LIN {X 0,Y 262.413,Z 305.616,A -85,B 0,C 180,E1 -18658.413,E2 -18658.413} C_VEL
LIN {X 0,Y 260.939,Z 356.529,A -85,B 0,C 180,E1 -18660.058,E2 -18660.058} C_VEL
LIN {X 0,Y 260.58,Z 366.415,A -85,B 0,C 180,E1 -18660.585,E2 -18660.585} C_VEL
LIN {X 0,Y 259.89,Z 377.928,A -85,B 0,C 180,E1 -18661.482,E2 -18661.482} C_VEL
LIN {X 0,Y 259.092,Z 388.369,A -85,B 0,C 180,E1 -18662.636,E2 -18662.636} C_VEL
LIN {X 0,Y 258.368,Z 397.253,A -85,B 0,C 180,E1 -18663.891,E2 -18663.891} C_VEL
LIN {X 0,Y 257.495,Z 404.951,A -85,B 0,C 180,E1 -18665.226,E2 -18665.226} C_VEL
LIN {X 0,Y 256.533,Z 413.514,A -85,B 0,C 180,E1 -18667.063,E2 -18667.063} C_VEL
LIN {X 0,Y 255.727,Z 421.136,A -85,B 0,C 180,E1 -18669.203,E2 -18669.203} C_VEL
LIN {X 0,Y 255.116,Z 426.116,A -85,B 0,C 180,E1 -18670.941,E2 -18670.941} C_VEL
LIN {X 0,Y 254.737,Z 430.48,A -85,B 0,C 180,E1 -18672.842,E2 -18672.842} C_VEL
LIN {X 0,Y 254.278,Z 434.421,A -85,B 0,C 180,E1 -18675.095,E2 -18675.095} C_VEL
LIN {X 0,Y 254.025,Z 437.165,A -85,B 0,C 180,E1 -18677.329,E2 -18677.329} C_VEL
LIN {X 0,Y 254.008,Z 438.048,A -85,B 0,C 180,E1 -18678.393,E2 -18678.393} C_VEL
LIN {X 0,Y 254.169,Z 439.211,A -85,B 0,C 180,E1 -18680.733,E2 -18680.733} C_VEL
LIN {X 0,Y 254.592,Z 439.262,A -85,B 0,C 180,E1 -18683.18,E2 -18683.18} C_VEL
LIN {X 0,Y 255.349,Z 438.101,A -85,B 0,C 180,E1 -18685.656,E2 -18685.656} C_VEL
LIN {X 0,Y 256.573,Z 434.825,A -85,B 0,C 180,E1 -18688.64,E2 -18688.64} C_VEL
LIN {X 0,Y 257.683,Z 431.567,A -85,B 0,C 180,E1 -18690.6,E2 -18690.6} C_VEL
LIN {X 0,Y 258.955,Z 427.356,A -85,B 0,C 180,E1 -18692.526,E2 -18692.526} C_VEL
LIN {X 0,Y 260.481,Z 422.037,A -85,B 0,C 180,E1 -18694.427,E2 -18694.427} C_VEL
LIN {X 0,Y 262.359,Z 415.32,A -85,B 0,C 180,E1 -18696.31,E2 -18696.31} C_VEL
LIN {X 0,Y 264.289,Z 406.845,A -85,B 0,C 180,E1 -18698.145,E2 -18698.145} C_VEL
LIN {X 0,Y 265.906,Z 399.02,A -85,B 0,C 180,E1 -18699.502,E2 -18699.502} C_VEL
LIN {X 0,Y 267.227,Z 391.67,A -85,B 0,C 180,E1 -18700.543,E2 -18700.543} C_VEL
LIN {X 0,Y 268.577,Z 382.564,A -85,B 0,C 180,E1 -18701.58,E2 -18701.58} C_VEL
LIN {X 0,Y 269.878,Z 372.132,A -85,B 0,C 180,E1 -18702.478,E2 -18702.478} C_VEL
LIN {X 0,Y 270.737,Z 360.477,A -85,B 0,C 180,E1 -18703.167,E2 -18703.167} C_VEL
LIN {X 0,Y 271.796,Z 338.049,A -85,B 0,C 180,E1 -18703.941,E2 -18703.941} C_VEL
LIN {X 0,Y 272.811,Z 314.84,A -85,B 0,C 180,E1 -18704.695,E2 -18704.695} C_VEL
LIN {X 0,Y 268.494,Z 305.093,A -85,B 0,C 180,E1 -18705.731,E2 -18705.731} C_VEL
LIN {X 0,Y 262.601,Z 294.531,A -85,B 0,C 180,E1 -18707.147,E2 -18707.147} C_VEL
LIN {X 0,Y 258.247,Z 287.429,A -85,B 0,C 180,E1 -18708.241,E2 -18708.241} C_VEL
LIN {X 0,Y 256.704,Z 285.058,A -85,B 0,C 180,E1 -18708.638,E2 -18708.638} C_VEL
LIN {X 0,Y 256.281,Z 283.378,A -85,B 0,C 180,E1 -18708.844,E2 -18708.844} C_VEL
LIN {X 0,Y 256.508,Z 283.344,A -85,B 0,C 180,E1 -18712.128,E2 -18712.128} C_VEL
LIN {X 0,Y 256.494,Z 283.345,A -85,B 0,C 180,E1 -18716.86,E2 -18716.86} C_VEL
LIN {X 0,Y 256.759,Z 283.312,A -85,B 0,C 180,E1 -18720.001,E2 -18720.001} C_VEL
LIN {X 0,Y 256.494,Z 283.347,A -85,B 0,C 180,E1 -18723.143,E2 -18723.143} C_VEL
LIN {X 0,Y 256.534,Z 283.334,A -85,B 0,C 180,E1 -18727.874,E2 -18727.874} C_VEL
LIN {X 0,Y 256.503,Z 283.337,A -85,B 0,C 180,E1 -18728.248,E2 -18728.248} C_VEL
LIN {X 0,Y 255.757,Z 283.436,A -85,B 0,C 180,E1 -18729.556,E2 -18729.556} C_VEL
LIN {X 0,Y 252.8,Z 283.81,A -85,B 0,C 180,E1 -18731.686,E2 -18731.686} C_VEL
LIN {X 0,Y 250.323,Z 284.12,A -85,B 0,C 180,E1 -18733.42,E2 -18733.42} C_VEL
LIN {X 0,Y 249.264,Z 284.248,A -85,B 0,C 180,E1 -18734.766,E2 -18734.766} C_VEL
LIN {X 0,Y 249.178,Z 284.253,A -85,B 0,C 180,E1 -18735.223,E2 -18735.223} C_VEL
LIN {X 0,Y 249.131,Z 284.26,A -85,B 0,C 180,E1 -18738.079,E2 -18738.079} C_VEL
LIN {X 0,Y 249.084,Z 284.258,A -85,B 0,C 180,E1 -18741.52,E2 -18741.52} C_VEL
LIN {X 0,Y 249.128,Z 284.252,A -85,B 0,C 180,E1 -18745.484,E2 -18745.484} C_VEL
LIN {X 0,Y 249.083,Z 284.259,A -85,B 0,C 180,E1 -18748.996,E2 -18748.996} C_VEL
LIN {X 0,Y 249.034,Z 284.271,A -85,B 0,C 180,E1 -18752.427,E2 -18752.427} C_VEL
LIN {X 0,Y 249.072,Z 284.267,A -85,B 0,C 180,E1 -18756.339,E2 -18756.339} C_VEL
LIN {X 0,Y 249.036,Z 284.27,A -85,B 0,C 180,E1 -18760.473,E2 -18760.473} C_VEL
LIN {X 0,Y 249.033,Z 284.276,A -85,B 0,C 180,E1 -18762.8,E2 -18762.8} C_VEL
LIN {X 0,Y 249.018,Z 284.277,A -85,B 0,C 180,E1 -18767.365,E2 -18767.365} C_VEL
LIN {X 0,Y 249.056,Z 284.41,A -85,B 0,C 180,E1 -18771.174,E2 -18771.174} C_VEL
LIN {X 0,Y 250.877,Z 290.539,A -85,B 0,C 180,E1 -18774.332,E2 -18774.332} C_VEL
LIN {X 0,Y 252.867,Z 298.716,A -85,B 0,C 180,E1 -18778.126,E2 -18778.126} C_VEL
LIN {X 0,Y 253.754,Z 302.564,A -85,B 0,C 180,E1 -18779.725,E2 -18779.725} C_VEL
LIN {X 0,Y 255.811,Z 306.867,A -85,B 0,C 180,E1 -18780.308,E2 -18780.308} C_VEL
LIN {X 0,Y 259.48,Z 315.185,A -85,B 0,C 180,E1 -18781.332,E2 -18781.332} C_VEL
LIN {X 0,Y 262.764,Z 332.237,A -85,B 0,C 180,E1 -18782.601,E2 -18782.601} C_VEL
LIN {X 0,Y 264.983,Z 349.14,A -85,B 0,C 180,E1 -18783.635,E2 -18783.635} C_VEL
LIN {X 0,Y 265.432,Z 356.335,A -85,B 0,C 180,E1 -18783.987,E2 -18783.987} C_VEL
LIN {X 0,Y 263.95,Z 383.888,A -85,B 0,C 180,E1 -18784.924,E2 -18784.924} C_VEL
LIN {X 0,Y 262.737,Z 395.64,A -85,B 0,C 180,E1 -18785.573,E2 -18785.573} C_VEL
LIN {X 0,Y 261.153,Z 405.827,A -85,B 0,C 180,E1 -18786.404,E2 -18786.404} C_VEL
LIN {X 0,Y 259.584,Z 414.308,A -85,B 0,C 180,E1 -18787.307,E2 -18787.307} C_VEL
LIN {X 0,Y 257.892,Z 422.523,A -85,B 0,C 180,E1 -18788.415,E2 -18788.415} C_VEL
LIN {X 0,Y 256.092,Z 430.382,A -85,B 0,C 180,E1 -18789.729,E2 -18789.729} C_VEL
LIN {X 0,Y 254.423,Z 436.939,A -85,B 0,C 180,E1 -18791.061,E2 -18791.061} C_VEL
LIN {X 0,Y 252.738,Z 443.225,A -85,B 0,C 180,E1 -18792.607,E2 -18792.607} C_VEL
LIN {X 0,Y 251.217,Z 448.504,A -85,B 0,C 180,E1 -18794.172,E2 -18794.172} C_VEL
LIN {X 0,Y 249.775,Z 453.917,A -85,B 0,C 180,E1 -18796.163,E2 -18796.163} C_VEL
LIN {X 0,Y 248.415,Z 459.006,A -85,B 0,C 180,E1 -18798.578,E2 -18798.578} C_VEL
LIN {X 0,Y 247.812,Z 461.526,A -85,B 0,C 180,E1 -18800.203,E2 -18800.203} C_VEL
LIN {X 0,Y 247.369,Z 463.503,A -85,B 0,C 180,E1 -18801.834,E2 -18801.834} C_VEL
LIN {X 0,Y 246.986,Z 465.878,A -85,B 0,C 180,E1 -18804.834,E2 -18804.834} C_VEL
LIN {X 0,Y 247.05,Z 466.43,A -85,B 0,C 180,E1 -18806.739,E2 -18806.739} C_VEL
LIN {X 0,Y 247.107,Z 466.306,A -85,B 0,C 180,E1 -18808.371,E2 -18808.371} C_VEL
LIN {X 0,Y 247.233,Z 465.701,A -85,B 0,C 180,E1 -18810,E2 -18810} C_VEL
LIN {X 0,Y 247.156,Z 464.577,A -85,B 0,C 180,E1 -18811.63,E2 -18811.63} C_VEL
LIN {X 0,Y 247.203,Z 462.925,A -85,B 0,C 180,E1 -18813.26,E2 -18813.26} C_VEL
LIN {X 0,Y 247.195,Z 459.237,A -85,B 0,C 180,E1 -18815.676,E2 -18815.676} C_VEL
LIN {X 0,Y 247.425,Z 453.965,A -85,B 0,C 180,E1 -18818.165,E2 -18818.165} C_VEL
LIN {X 0,Y 247.837,Z 448.329,A -85,B 0,C 180,E1 -18820.209,E2 -18820.209} C_VEL
LIN {X 0,Y 248.555,Z 441.204,A -85,B 0,C 180,E1 -18822.244,E2 -18822.244} C_VEL
LIN {X 0,Y 249.399,Z 433.015,A -85,B 0,C 180,E1 -18824.067,E2 -18824.067} C_VEL
LIN {X 0,Y 250.162,Z 426.449,A -85,B 0,C 180,E1 -18825.271,E2 -18825.271} C_VEL
LIN {X 0,Y 250.921,Z 420.034,A -85,B 0,C 180,E1 -18826.266,E2 -18826.266} C_VEL
LIN {X 0,Y 251.602,Z 412.242,A -85,B 0,C 180,E1 -18827.265,E2 -18827.265} C_VEL
LIN {X 0,Y 252.641,Z 402.367,A -85,B 0,C 180,E1 -18828.237,E2 -18828.237} C_VEL
LIN {X 0,Y 253.32,Z 393.113,A -85,B 0,C 180,E1 -18828.92,E2 -18828.92} C_VEL
LIN {X 0,Y 253.729,Z 383.59,A -85,B 0,C 180,E1 -18829.414,E2 -18829.414} C_VEL
LIN {X 0,Y 254.605,Z 351.161,A -85,B 0,C 180,E1 -18830.505,E2 -18830.505} C_VEL
LIN {X 0,Y 250.337,Z 306.801,A -85,B 0,C 180,E1 -18832.309,E2 -18832.309} C_VEL
LIN {X 0,Y 251.565,Z 297.448,A -85,B 0,C 180,E1 -18835.66,E2 -18835.66} C_VEL
LIN {X 0,Y 249.84,Z 287.931,A -85,B 0,C 180,E1 -18839.303,E2 -18839.303} C_VEL
LIN {X 0,Y 249.12,Z 284.266,A -85,B 0,C 180,E1 -18840.752,E2 -18840.752} C_VEL
LIN {X 0,Y 249.052,Z 284.273,A -85,B 0,C 180,E1 -18845.079,E2 -18845.079} C_VEL
LIN {X 0,Y 249.04,Z 284.274,A -85,B 0,C 180,E1 -18848.378,E2 -18848.378} C_VEL
LIN {X 0,Y 249.014,Z 284.275,A -85,B 0,C 180,E1 -18852.792,E2 -18852.792} C_VEL
LIN {X 0,Y 249.011,Z 284.28,A -85,B 0,C 180,E1 -18857.36,E2 -18857.36} C_VEL
LIN {X 0,Y 249.026,Z 284.277,A -85,B 0,C 180,E1 -18861.618,E2 -18861.618} C_VEL
LIN {X 0,Y 249.044,Z 284.277,A -85,B 0,C 180,E1 -18865.638,E2 -18865.638} C_VEL
LIN {X 0,Y 249.052,Z 284.274,A -85,B 0,C 180,E1 -18869.472,E2 -18869.472} C_VEL
LIN {X 0,Y 249.074,Z 284.271,A -85,B 0,C 180,E1 -18873.161,E2 -18873.161} C_VEL
LIN {X 0,Y 249.079,Z 284.268,A -85,B 0,C 180,E1 -18876.731,E2 -18876.731} C_VEL
LIN {X 0,Y 249.11,Z 284.265,A -85,B 0,C 180,E1 -18880.21,E2 -18880.21} C_VEL
LIN {X 0,Y 249.241,Z 284.253,A -85,B 0,C 180,E1 -18883.621,E2 -18883.621} C_VEL
LIN {X 0,Y 249.242,Z 284.247,A -85,B 0,C 180,E1 -18888.615,E2 -18888.615} C_VEL
LIN {X 0,Y 249.453,Z 284.224,A -85,B 0,C 180,E1 -18891.901,E2 -18891.901} C_VEL
LIN {X 0,Y 249.294,Z 284.241,A -85,B 0,C 180,E1 -18895.147,E2 -18895.147} C_VEL
LIN {X 0,Y 249.673,Z 284.195,A -85,B 0,C 180,E1 -18898.386,E2 -18898.386} C_VEL
LIN {X 0,Y 249.673,Z 284.199,A -85,B 0,C 180,E1 -18901.612,E2 -18901.612} C_VEL
LIN {X 0,Y 249.446,Z 284.221,A -85,B 0,C 180,E1 -18906.773,E2 -18906.773} C_VEL
LIN {X 0,Y 249.385,Z 284.234,A -85,B 0,C 180,E1 -18909.733,E2 -18909.733} C_VEL
LIN {X 0,Y 249.197,Z 284.253,A -85,B 0,C 180,E1 -18914.702,E2 -18914.702} C_VEL
LIN {X 0,Y 249.135,Z 284.263,A -85,B 0,C 180,E1 -18918.076,E2 -18918.076} C_VEL
LIN {X 0,Y 249.099,Z 284.267,A -85,B 0,C 180,E1 -18921.515,E2 -18921.515} C_VEL
LIN {X 0,Y 249.125,Z 284.266,A -85,B 0,C 180,E1 -18925.481,E2 -18925.481} C_VEL
LIN {X 0,Y 249.075,Z 284.268,A -85,B 0,C 180,E1 -18928.991,E2 -18928.991} C_VEL
LIN {X 0,Y 249.03,Z 284.275,A -85,B 0,C 180,E1 -18932.424,E2 -18932.424} C_VEL
LIN {X 0,Y 249.07,Z 284.269,A -85,B 0,C 180,E1 -18936.337,E2 -18936.337} C_VEL
LIN {X 0,Y 249.032,Z 284.275,A -85,B 0,C 180,E1 -18940.471,E2 -18940.471} C_VEL
LIN {X 0,Y 249.042,Z 284.273,A -85,B 0,C 180,E1 -18942.801,E2 -18942.801} C_VEL
LIN {X 0,Y 249.056,Z 284.271,A -85,B 0,C 180,E1 -18947.372,E2 -18947.372} C_VEL
LIN {X 0,Y 249.046,Z 284.277,A -85,B 0,C 180,E1 -18951.623,E2 -18951.623} C_VEL
LIN {X 0,Y 249.055,Z 284.273,A -85,B 0,C 180,E1 -18955.642,E2 -18955.642} C_VEL
LIN {X 0,Y 249.045,Z 284.275,A -85,B 0,C 180,E1 -18959.472,E2 -18959.472} C_VEL
LIN {X 0,Y 249.067,Z 284.269,A -85,B 0,C 180,E1 -18963.162,E2 -18963.162} C_VEL
LIN {X 0,Y 249.072,Z 284.27,A -85,B 0,C 180,E1 -18966.732,E2 -18966.732} C_VEL
LIN {X 0,Y 249.103,Z 284.266,A -85,B 0,C 180,E1 -18970.211,E2 -18970.211} C_VEL
LIN {X 0,Y 249.235,Z 284.251,A -85,B 0,C 180,E1 -18973.621,E2 -18973.621} C_VEL
LIN {X 0,Y 249.246,Z 284.247,A -85,B 0,C 180,E1 -18978.616,E2 -18978.616} C_VEL
LIN {X 0,Y 249.474,Z 284.223,A -85,B 0,C 180,E1 -18981.902,E2 -18981.902} C_VEL
LIN {X 0,Y 249.426,Z 284.225,A -85,B 0,C 180,E1 -18986.769,E2 -18986.769} C_VEL
LIN {X 0,Y 249.72,Z 284.191,A -85,B 0,C 180,E1 -18990,E2 -18990} C_VEL
LIN {X 0,Y 249.426,Z 284.226,A -85,B 0,C 180,E1 -18993.23,E2 -18993.23} C_VEL
LIN {X 0,Y 249.472,Z 284.221,A -85,B 0,C 180,E1 -18998.097,E2 -18998.097} C_VEL
LIN {X 0,Y 249.245,Z 284.249,A -85,B 0,C 180,E1 -19001.383,E2 -19001.383} C_VEL
LIN {X 0,Y 249.234,Z 284.251,A -85,B 0,C 180,E1 -19006.378,E2 -19006.378} C_VEL
LIN {X 0,Y 249.076,Z 284.272,A -85,B 0,C 180,E1 -19011.518,E2 -19011.518} C_VEL
LIN {X 0,Y 249.112,Z 284.267,A -85,B 0,C 180,E1 -19015.477,E2 -19015.477} C_VEL
LIN {X 0,Y 249.137,Z 284.413,A -85,B 0,C 180,E1 -19016.89,E2 -19016.89} C_VEL
LIN {X 0,Y 255.379,Z 303.773,A -85,B 0,C 180,E1 -19017.949,E2 -19017.949} C_VEL
LIN {X 0,Y 255.335,Z 313.119,A -85,B 0,C 180,E1 -19018.266,E2 -19018.266} C_VEL
LIN {X 0,Y 253.983,Z 356.955,A -85,B 0,C 180,E1 -19019.729,E2 -19019.729} C_VEL
LIN {X 0,Y 253.595,Z 367.606,A -85,B 0,C 180,E1 -19020.321,E2 -19020.321} C_VEL
LIN {X 0,Y 252.936,Z 378.268,A -85,B 0,C 180,E1 -19021.188,E2 -19021.188} C_VEL
LIN {X 0,Y 252.224,Z 387.215,A -85,B 0,C 180,E1 -19022.173,E2 -19022.173} C_VEL
LIN {X 0,Y 251.439,Z 396.631,A -85,B 0,C 180,E1 -19023.503,E2 -19023.503} C_VEL
LIN {X 0,Y 250.641,Z 403.843,A -85,B 0,C 180,E1 -19024.749,E2 -19024.749} C_VEL
LIN {X 0,Y 249.787,Z 410.867,A -85,B 0,C 180,E1 -19026.216,E2 -19026.216} C_VEL
LIN {X 0,Y 249.097,Z 417.185,A -85,B 0,C 180,E1 -19027.818,E2 -19027.818} C_VEL
LIN {X 0,Y 248.377,Z 423.251,A -85,B 0,C 180,E1 -19029.694,E2 -19029.694} C_VEL
LIN {X 0,Y 247.772,Z 429.196,A -85,B 0,C 180,E1 -19032.015,E2 -19032.015} C_VEL
LIN {X 0,Y 247.392,Z 432.744,A -85,B 0,C 180,E1 -19033.825,E2 -19033.825} C_VEL
LIN {X 0,Y 247.157,Z 435.002,A -85,B 0,C 180,E1 -19035.305,E2 -19035.305} C_VEL
LIN {X 0,Y 246.912,Z 437.829,A -85,B 0,C 180,E1 -19037.734,E2 -19037.734} C_VEL
LIN {X 0,Y 247.024,Z 439.415,A -85,B 0,C 180,E1 -19040.188,E2 -19040.188} C_VEL
LIN {X 0,Y 247.552,Z 439.696,A -85,B 0,C 180,E1 -19043.405,E2 -19043.405} C_VEL
LIN {X 0,Y 248.2,Z 438.833,A -85,B 0,C 180,E1 -19045.508,E2 -19045.508} C_VEL
LIN {X 0,Y 249.12,Z 436.904,A -85,B 0,C 180,E1 -19047.813,E2 -19047.813} C_VEL
LIN {X 0,Y 250.496,Z 433.299,A -85,B 0,C 180,E1 -19050.426,E2 -19050.426} C_VEL
LIN {X 0,Y 251.767,Z 429.419,A -85,B 0,C 180,E1 -19052.413,E2 -19052.413} C_VEL
LIN {X 0,Y 253.445,Z 423.975,A -85,B 0,C 180,E1 -19054.546,E2 -19054.546} C_VEL
LIN {X 0,Y 254.957,Z 418.94,A -85,B 0,C 180,E1 -19056.118,E2 -19056.118} C_VEL
LIN {X 0,Y 256.614,Z 412.846,A -85,B 0,C 180,E1 -19057.68,E2 -19057.68} C_VEL
LIN {X 0,Y 258.212,Z 406.364,A -85,B 0,C 180,E1 -19059.046,E2 -19059.046} C_VEL
LIN {X 0,Y 259.864,Z 398.652,A -85,B 0,C 180,E1 -19060.382,E2 -19060.382} C_VEL
LIN {X 0,Y 261.442,Z 390.014,A -85,B 0,C 180,E1 -19061.589,E2 -19061.589} C_VEL
LIN {X 0,Y 263.194,Z 378.281,A -85,B 0,C 180,E1 -19062.82,E2 -19062.82} C_VEL
LIN {X 0,Y 264.216,Z 367.992,A -85,B 0,C 180,E1 -19063.598,E2 -19063.598} C_VEL
LIN {X 0,Y 264.948,Z 358.296,A -85,B 0,C 180,E1 -19064.098,E2 -19064.098} C_VEL
LIN {X 0,Y 266.9,Z 316.919,A -85,B 0,C 180,E1 -19065.501,E2 -19065.501} C_VEL
LIN {X 0,Y 263.411,Z 308.95,A -85,B 0,C 180,E1 -19066.403,E2 -19066.403} C_VEL
LIN {X 0,Y 257.551,Z 298.407,A -85,B 0,C 180,E1 -19067.877,E2 -19067.877} C_VEL
LIN {X 0,Y 253.374,Z 291.754,A -85,B 0,C 180,E1 -19068.983,E2 -19068.983} C_VEL
LIN {X 0,Y 251.406,Z 288.478,A -85,B 0,C 180,E1 -19069.533,E2 -19069.533} C_VEL
LIN {X 0,Y 249.771,Z 285.962,A -85,B 0,C 180,E1 -19069.996,E2 -19069.996} C_VEL
LIN {X 0,Y 249.357,Z 284.236,A -85,B 0,C 180,E1 -19070.215,E2 -19070.215} C_VEL
LIN {X 0,Y 249.447,Z 284.228,A -85,B 0,C 180,E1 -19073.531,E2 -19073.531} C_VEL
LIN {X 0,Y 249.67,Z 284.193,A -85,B 0,C 180,E1 -19078.388,E2 -19078.388} C_VEL
LIN {X 0,Y 249.67,Z 284.191,A -85,B 0,C 180,E1 -19081.614,E2 -19081.614} C_VEL
LIN {X 0,Y 249.455,Z 284.226,A -85,B 0,C 180,E1 -19086.472,E2 -19086.472} C_VEL
LIN {X 0,Y 249.384,Z 284.232,A -85,B 0,C 180,E1 -19089.736,E2 -19089.736} C_VEL
LIN {X 0,Y 249.193,Z 284.257,A -85,B 0,C 180,E1 -19094.705,E2 -19094.705} C_VEL
LIN {X 0,Y 249.178,Z 284.253,A -85,B 0,C 180,E1 -19095.223,E2 -19095.223} C_VEL
LIN {X 0,Y 248.502,Z 284.332,A -85,B 0,C 180,E1 -19096.571,E2 -19096.571} C_VEL
LIN {X 0,Y 245.618,Z 284.702,A -85,B 0,C 180,E1 -19098.767,E2 -19098.767} C_VEL
LIN {X 0,Y 243.16,Z 285.008,A -85,B 0,C 180,E1 -19100.555,E2 -19100.555} C_VEL
LIN {X 0,Y 242.095,Z 285.134,A -85,B 0,C 180,E1 -19101.943,E2 -19101.943} C_VEL
LIN {X 0,Y 242.002,Z 285.144,A -85,B 0,C 180,E1 -19102.414,E2 -19102.414} C_VEL
LIN {X 0,Y 242.064,Z 285.133,A -85,B 0,C 180,E1 -19105.84,E2 -19105.84} C_VEL
LIN {X 0,Y 242.029,Z 285.137,A -85,B 0,C 180,E1 -19109.582,E2 -19109.582} C_VEL
LIN {X 0,Y 241.989,Z 285.143,A -85,B 0,C 180,E1 -19113.493,E2 -19113.493} C_VEL
LIN {X 0,Y 242.009,Z 285.143,A -85,B 0,C 180,E1 -19117.58,E2 -19117.58} C_VEL
LIN {X 0,Y 241.96,Z 285.158,A -85,B 0,C 180,E1 -19121.919,E2 -19121.919} C_VEL
LIN {X 0,Y 241.937,Z 285.156,A -85,B 0,C 180,E1 -19126.572,E2 -19126.572} C_VEL
LIN {X 0,Y 241.989,Z 285.359,A -85,B 0,C 180,E1 -19129.812,E2 -19129.812} C_VEL
LIN {X 0,Y 244.398,Z 293.32,A -85,B 0,C 180,E1 -19134.17,E2 -19134.17} C_VEL
LIN {X 0,Y 246.442,Z 301.873,A -85,B 0,C 180,E1 -19138.198,E2 -19138.198} C_VEL
LIN {X 0,Y 252.059,Z 313.372,A -85,B 0,C 180,E1 -19139.894,E2 -19139.894} C_VEL
LIN {X 0,Y 254.241,Z 318.686,A -85,B 0,C 180,E1 -19140.55,E2 -19140.55} C_VEL
LIN {X 0,Y 257.29,Z 334.984,A -85,B 0,C 180,E1 -19141.802,E2 -19141.802} C_VEL
LIN {X 0,Y 259.369,Z 352.201,A -85,B 0,C 180,E1 -19142.88,E2 -19142.88} C_VEL
LIN {X 0,Y 259.575,Z 357.239,A -85,B 0,C 180,E1 -19143.125,E2 -19143.125} C_VEL
LIN {X 0,Y 258.032,Z 383.822,A -85,B 0,C 180,E1 -19144.06,E2 -19144.06} C_VEL
LIN {X 0,Y 256.733,Z 395.495,A -85,B 0,C 180,E1 -19144.728,E2 -19144.728} C_VEL
LIN {X 0,Y 255.075,Z 405.756,A -85,B 0,C 180,E1 -19145.589,E2 -19145.589} C_VEL
LIN {X 0,Y 253.425,Z 414.174,A -85,B 0,C 180,E1 -19146.507,E2 -19146.507} C_VEL
LIN {X 0,Y 251.644,Z 422.342,A -85,B 0,C 180,E1 -19147.635,E2 -19147.635} C_VEL
LIN {X 0,Y 249.756,Z 430.165,A -85,B 0,C 180,E1 -19148.976,E2 -19148.976} C_VEL
LIN {X 0,Y 247.753,Z 437.555,A -85,B 0,C 180,E1 -19150.531,E2 -19150.531} C_VEL
LIN {X 0,Y 245.573,Z 445.112,A -85,B 0,C 180,E1 -19152.513,E2 -19152.513} C_VEL
LIN {X 0,Y 243.418,Z 452.074,A -85,B 0,C 180,E1 -19154.94,E2 -19154.94} C_VEL
LIN {X 0,Y 241.857,Z 457.428,A -85,B 0,C 180,E1 -19157.413,E2 -19157.413} C_VEL
LIN {X 0,Y 240.785,Z 461.439,A -85,B 0,C 180,E1 -19159.915,E2 -19159.915} C_VEL
LIN {X 0,Y 240.326,Z 463.323,A -85,B 0,C 180,E1 -19161.593,E2 -19161.593} C_VEL
LIN {X 0,Y 240.033,Z 464.71,A -85,B 0,C 180,E1 -19163.275,E2 -19163.275} C_VEL
LIN {X 0,Y 239.923,Z 465.624,A -85,B 0,C 180,E1 -19164.959,E2 -19164.959} C_VEL
LIN {X 0,Y 239.962,Z 466.046,A -85,B 0,C 180,E1 -19166.642,E2 -19166.642} C_VEL
LIN {X 0,Y 240.032,Z 465.859,A -85,B 0,C 180,E1 -19168.323,E2 -19168.323} C_VEL
LIN {X 0,Y 240.152,Z 465.168,A -85,B 0,C 180,E1 -19170,E2 -19170} C_VEL
LIN {X 0,Y 240.084,Z 463.96,A -85,B 0,C 180,E1 -19171.678,E2 -19171.678} C_VEL
LIN {X 0,Y 240.141,Z 462.229,A -85,B 0,C 180,E1 -19173.356,E2 -19173.356} C_VEL
LIN {X 0,Y 240.109,Z 458.853,A -85,B 0,C 180,E1 -19175.618,E2 -19175.618} C_VEL
LIN {X 0,Y 240.274,Z 455.021,A -85,B 0,C 180,E1 -19177.564,E2 -19177.564} C_VEL
LIN {X 0,Y 240.541,Z 450.917,A -85,B 0,C 180,E1 -19179.248,E2 -19179.248} C_VEL
LIN {X 0,Y 240.935,Z 445.938,A -85,B 0,C 180,E1 -19180.93,E2 -19180.93} C_VEL
LIN {X 0,Y 241.564,Z 439.923,A -85,B 0,C 180,E1 -19182.604,E2 -19182.604} C_VEL
LIN {X 0,Y 242.361,Z 432.591,A -85,B 0,C 180,E1 -19184.27,E2 -19184.27} C_VEL
LIN {X 0,Y 243.145,Z 426.019,A -85,B 0,C 180,E1 -19185.508,E2 -19185.508} C_VEL
LIN {X 0,Y 243.919,Z 419.593,A -85,B 0,C 180,E1 -19186.531,E2 -19186.531} C_VEL
LIN {X 0,Y 244.628,Z 411.791,A -85,B 0,C 180,E1 -19187.557,E2 -19187.557} C_VEL
LIN {X 0,Y 245.692,Z 401.906,A -85,B 0,C 180,E1 -19188.556,E2 -19188.556} C_VEL
LIN {X 0,Y 246.39,Z 392.639,A -85,B 0,C 180,E1 -19189.257,E2 -19189.257} C_VEL
LIN {X 0,Y 246.821,Z 383.1,A -85,B 0,C 180,E1 -19189.763,E2 -19189.763} C_VEL
LIN {X 0,Y 247.676,Z 351.616,A -85,B 0,C 180,E1 -19190.856,E2 -19190.856} C_VEL
LIN {X 0,Y 243.387,Z 306.47,A -85,B 0,C 180,E1 -19192.731,E2 -19192.731} C_VEL
LIN {X 0,Y 244.5,Z 298.832,A -85,B 0,C 180,E1 -19195.541,E2 -19195.541} C_VEL
LIN {X 0,Y 243.779,Z 293.87,A -85,B 0,C 180,E1 -19197.469,E2 -19197.469} C_VEL
LIN {X 0,Y 242.072,Z 285.146,A -85,B 0,C 180,E1 -19201.019,E2 -19201.019} C_VEL
LIN {X 0,Y 242.009,Z 285.152,A -85,B 0,C 180,E1 -19205.596,E2 -19205.596} C_VEL
LIN {X 0,Y 241.976,Z 285.156,A -85,B 0,C 180,E1 -19209.715,E2 -19209.715} C_VEL
LIN {X 0,Y 241.929,Z 285.159,A -85,B 0,C 180,E1 -19214.202,E2 -19214.202} C_VEL
LIN {X 0,Y 241.935,Z 285.16,A -85,B 0,C 180,E1 -19218.076,E2 -19218.076} C_VEL
LIN {X 0,Y 241.99,Z 285.15,A -85,B 0,C 180,E1 -19222.417,E2 -19222.417} C_VEL
LIN {X 0,Y 241.981,Z 285.153,A -85,B 0,C 180,E1 -19226.506,E2 -19226.506} C_VEL
LIN {X 0,Y 242.038,Z 285.144,A -85,B 0,C 180,E1 -19230.586,E2 -19230.586} C_VEL
LIN {X 0,Y 242.068,Z 285.143,A -85,B 0,C 180,E1 -19234.182,E2 -19234.182} C_VEL
LIN {X 0,Y 242.053,Z 285.142,A -85,B 0,C 180,E1 -19238.296,E2 -19238.296} C_VEL
LIN {X 0,Y 242.163,Z 285.132,A -85,B 0,C 180,E1 -19243.277,E2 -19243.277} C_VEL
LIN {X 0,Y 242.179,Z 285.128,A -85,B 0,C 180,E1 -19248.278,E2 -19248.278} C_VEL
LIN {X 0,Y 242.398,Z 285.105,A -85,B 0,C 180,E1 -19251.663,E2 -19251.663} C_VEL
LIN {X 0,Y 242.255,Z 285.118,A -85,B 0,C 180,E1 -19255.006,E2 -19255.006} C_VEL
LIN {X 0,Y 242.633,Z 285.072,A -85,B 0,C 180,E1 -19258.339,E2 -19258.339} C_VEL
LIN {X 0,Y 242.633,Z 285.075,A -85,B 0,C 180,E1 -19261.658,E2 -19261.658} C_VEL
LIN {X 0,Y 242.424,Z 285.097,A -85,B 0,C 180,E1 -19266.751,E2 -19266.751} C_VEL
LIN {X 0,Y 242.311,Z 285.113,A -85,B 0,C 180,E1 -19270.02,E2 -19270.02} C_VEL
LIN {X 0,Y 242.16,Z 285.131,A -85,B 0,C 180,E1 -19275.14,E2 -19275.14} C_VEL
LIN {X 0,Y 242.075,Z 285.141,A -85,B 0,C 180,E1 -19278.622,E2 -19278.622} C_VEL
LIN {X 0,Y 242.045,Z 285.145,A -85,B 0,C 180,E1 -19282.175,E2 -19282.175} C_VEL
LIN {X 0,Y 242.062,Z 285.146,A -85,B 0,C 180,E1 -19285.837,E2 -19285.837} C_VEL
LIN {X 0,Y 242.024,Z 285.149,A -85,B 0,C 180,E1 -19289.579,E2 -19289.579} C_VEL
LIN {X 0,Y 241.986,Z 285.155,A -85,B 0,C 180,E1 -19293.49,E2 -19293.49} C_VEL
LIN {X 0,Y 242.006,Z 285.152,A -85,B 0,C 180,E1 -19297.577,E2 -19297.577} C_VEL
LIN {X 0,Y 241.963,Z 285.158,A -85,B 0,C 180,E1 -19301.915,E2 -19301.915} C_VEL
LIN {X 0,Y 241.985,Z 285.15,A -85,B 0,C 180,E1 -19306.556,E2 -19306.556} C_VEL
LIN {X 0,Y 242.001,Z 285.151,A -85,B 0,C 180,E1 -19310.29,E2 -19310.29} C_VEL
LIN {X 0,Y 242.03,Z 285.144,A -85,B 0,C 180,E1 -19314.497,E2 -19314.497} C_VEL
LIN {X 0,Y 241.969,Z 285.155,A -85,B 0,C 180,E1 -19318.479,E2 -19318.479} C_VEL
LIN {X 0,Y 242.002,Z 285.149,A -85,B 0,C 180,E1 -19322.312,E2 -19322.312} C_VEL
LIN {X 0,Y 242.05,Z 285.147,A -85,B 0,C 180,E1 -19326.015,E2 -19326.015} C_VEL
LIN {X 0,Y 242.031,Z 285.15,A -85,B 0,C 180,E1 -19329.607,E2 -19329.607} C_VEL
LIN {X 0,Y 242.156,Z 285.131,A -85,B 0,C 180,E1 -19333.278,E2 -19333.278} C_VEL
LIN {X 0,Y 242.179,Z 285.128,A -85,B 0,C 180,E1 -19338.279,E2 -19338.279} C_VEL
LIN {X 0,Y 242.42,Z 285.1,A -85,B 0,C 180,E1 -19341.665,E2 -19341.665} C_VEL
LIN {X 0,Y 242.25,Z 285.12,A -85,B 0,C 180,E1 -19345.007,E2 -19345.007} C_VEL
LIN {X 0,Y 242.628,Z 285.071,A -85,B 0,C 180,E1 -19348.34,E2 -19348.34} C_VEL
LIN {X 0,Y 242.628,Z 285.075,A -85,B 0,C 180,E1 -19351.659,E2 -19351.659} C_VEL
LIN {X 0,Y 242.423,Z 285.096,A -85,B 0,C 180,E1 -19356.659,E2 -19356.659} C_VEL
LIN {X 0,Y 242.306,Z 285.115,A -85,B 0,C 180,E1 -19360.021,E2 -19360.021} C_VEL
LIN {X 0,Y 242.159,Z 285.13,A -85,B 0,C 180,E1 -19365.141,E2 -19365.141} C_VEL
LIN {X 0,Y 242.064,Z 285.142,A -85,B 0,C 180,E1 -19368.624,E2 -19368.624} C_VEL
LIN {X 0,Y 241.998,Z 285.153,A -85,B 0,C 180,E1 -19372.18,E2 -19372.18} C_VEL
LIN {X 0,Y 242.06,Z 285.145,A -85,B 0,C 180,E1 -19376.454,E2 -19376.454} C_VEL
LIN {X 0,Y 248.556,Z 305.138,A -85,B 0,C 180,E1 -19377.586,E2 -19377.586} C_VEL
LIN {X 0,Y 247.954,Z 328.907,A -85,B 0,C 180,E1 -19378.389,E2 -19378.389} C_VEL
LIN {X 0,Y 247.04,Z 358.059,A -85,B 0,C 180,E1 -19379.417,E2 -19379.417} C_VEL
LIN {X 0,Y 246.65,Z 368.459,A -85,B 0,C 180,E1 -19380.027,E2 -19380.027} C_VEL
LIN {X 0,Y 245.889,Z 379.432,A -85,B 0,C 180,E1 -19380.971,E2 -19380.971} C_VEL
LIN {X 0,Y 245.133,Z 388.818,A -85,B 0,C 180,E1 -19382.067,E2 -19382.067} C_VEL
LIN {X 0,Y 244.403,Z 397.527,A -85,B 0,C 180,E1 -19383.356,E2 -19383.356} C_VEL
LIN {X 0,Y 243.458,Z 405.567,A -85,B 0,C 180,E1 -19384.819,E2 -19384.819} C_VEL
LIN {X 0,Y 242.456,Z 413.758,A -85,B 0,C 180,E1 -19386.66,E2 -19386.66} C_VEL
LIN {X 0,Y 241.712,Z 420.606,A -85,B 0,C 180,E1 -19388.606,E2 -19388.606} C_VEL
LIN {X 0,Y 240.977,Z 426.413,A -85,B 0,C 180,E1 -19390.69,E2 -19390.69} C_VEL
LIN {X 0,Y 240.64,Z 429.922,A -85,B 0,C 180,E1 -19392.199,E2 -19392.199} C_VEL
LIN {X 0,Y 240.16,Z 434.226,A -85,B 0,C 180,E1 -19394.613,E2 -19394.613} C_VEL
LIN {X 0,Y 239.843,Z 437.385,A -85,B 0,C 180,E1 -19397.1,E2 -19397.1} C_VEL
LIN {X 0,Y 239.91,Z 439.556,A -85,B 0,C 180,E1 -19399.876,E2 -19399.876} C_VEL
LIN {X 0,Y 240.232,Z 440.259,A -85,B 0,C 180,E1 -19402.173,E2 -19402.173} C_VEL
LIN {X 0,Y 240.851,Z 439.854,A -85,B 0,C 180,E1 -19404.787,E2 -19404.787} C_VEL
LIN {X 0,Y 241.46,Z 438.982,A -85,B 0,C 180,E1 -19406.428,E2 -19406.428} C_VEL
LIN {X 0,Y 242.359,Z 437.097,A -85,B 0,C 180,E1 -19408.538,E2 -19408.538} C_VEL
LIN {X 0,Y 243.503,Z 434.347,A -85,B 0,C 180,E1 -19410.618,E2 -19410.618} C_VEL
LIN {X 0,Y 245.309,Z 429.298,A -85,B 0,C 180,E1 -19413.273,E2 -19413.273} C_VEL
LIN {X 0,Y 246.882,Z 424.565,A -85,B 0,C 180,E1 -19415.162,E2 -19415.162} C_VEL
LIN {X 0,Y 248.371,Z 419.934,A -85,B 0,C 180,E1 -19416.664,E2 -19416.664} C_VEL
LIN {X 0,Y 250.138,Z 413.817,A -85,B 0,C 180,E1 -19418.293,E2 -19418.293} C_VEL
LIN {X 0,Y 251.977,Z 406.806,A -85,B 0,C 180,E1 -19419.81,E2 -19419.81} C_VEL
LIN {X 0,Y 253.729,Z 399.001,A -85,B 0,C 180,E1 -19421.189,E2 -19421.189} C_VEL
LIN {X 0,Y 255.56,Z 389.53,A -85,B 0,C 180,E1 -19422.528,E2 -19422.528} C_VEL
LIN {X 0,Y 257.238,Z 378.654,A -85,B 0,C 180,E1 -19423.674,E2 -19423.674} C_VEL
LIN {X 0,Y 258.315,Z 368.643,A -85,B 0,C 180,E1 -19424.451,E2 -19424.451} C_VEL
LIN {X 0,Y 259.085,Z 359.21,A -85,B 0,C 180,E1 -19424.956,E2 -19424.956} C_VEL
LIN {X 0,Y 261.207,Z 319.269,A -85,B 0,C 180,E1 -19426.335,E2 -19426.335} C_VEL
LIN {X 0,Y 257.866,Z 311.871,A -85,B 0,C 180,E1 -19427.229,E2 -19427.229} C_VEL
LIN {X 0,Y 251.577,Z 300.598,A -85,B 0,C 180,E1 -19428.929,E2 -19428.929} C_VEL
LIN {X 0,Y 247.006,Z 293.35,A -85,B 0,C 180,E1 -19430.224,E2 -19430.224} C_VEL
LIN {X 0,Y 244.591,Z 289.467,A -85,B 0,C 180,E1 -19430.958,E2 -19430.958} C_VEL
LIN {X 0,Y 242.915,Z 287.053,A -85,B 0,C 180,E1 -19431.474,E2 -19431.474} C_VEL
LIN {X 0,Y 242.411,Z 285.101,A -85,B 0,C 180,E1 -19431.771,E2 -19431.771} C_VEL
LIN {X 0,Y 242.253,Z 285.117,A -85,B 0,C 180,E1 -19435.009,E2 -19435.009} C_VEL
LIN {X 0,Y 242.63,Z 285.069,A -85,B 0,C 180,E1 -19438.342,E2 -19438.342} C_VEL
LIN {X 0,Y 242.631,Z 285.068,A -85,B 0,C 180,E1 -19441.661,E2 -19441.661} C_VEL
LIN {X 0,Y 242.428,Z 285.1,A -85,B 0,C 180,E1 -19446.66,E2 -19446.66} C_VEL
LIN {X 0,Y 242.309,Z 285.114,A -85,B 0,C 180,E1 -19450.023,E2 -19450.023} C_VEL
LIN {X 0,Y 242.149,Z 285.132,A -85,B 0,C 180,E1 -19455.205,E2 -19455.205} C_VEL
LIN {X 0,Y 242.067,Z 285.144,A -85,B 0,C 180,E1 -19458.626,E2 -19458.626} C_VEL
LIN {X 0,Y 242.002,Z 285.144,A -85,B 0,C 180,E1 -19462.414,E2 -19462.414} C_VEL
LIN {X 0,Y 241.306,Z 285.235,A -85,B 0,C 180,E1 -19463.803,E2 -19463.803} C_VEL
LIN {X 0,Y 238.419,Z 285.588,A -85,B 0,C 180,E1 -19466.067,E2 -19466.067} C_VEL
LIN {X 0,Y 236.01,Z 285.897,A -85,B 0,C 180,E1 -19467.913,E2 -19467.913} C_VEL
LIN {X 0,Y 235.023,Z 286.01,A -85,B 0,C 180,E1 -19469.346,E2 -19469.346} C_VEL
LIN {X 0,Y 234.967,Z 286.017,A -85,B 0,C 180,E1 -19469.831,E2 -19469.831} C_VEL
LIN {X 0,Y 234.959,Z 286.025,A -85,B 0,C 180,E1 -19474.635,E2 -19474.635} C_VEL
LIN {X 0,Y 234.941,Z 286.034,A -85,B 0,C 180,E1 -19478.946,E2 -19478.946} C_VEL
LIN {X 0,Y 234.927,Z 286.028,A -85,B 0,C 180,E1 -19483.478,E2 -19483.478} C_VEL
LIN {X 0,Y 234.909,Z 286.076,A -85,B 0,C 180,E1 -19488.163,E2 -19488.163} C_VEL
LIN {X 0,Y 236.836,Z 292.384,A -85,B 0,C 180,E1 -19491.948,E2 -19491.948} C_VEL
LIN {X 0,Y 238.313,Z 297.88,A -85,B 0,C 180,E1 -19494.896,E2 -19494.896} C_VEL
LIN {X 0,Y 239.164,Z 301.298,A -85,B 0,C 180,E1 -19496.506,E2 -19496.506} C_VEL
LIN {X 0,Y 241.616,Z 305.934,A -85,B 0,C 180,E1 -19497.331,E2 -19497.331} C_VEL
LIN {X 0,Y 245.372,Z 313.475,A -85,B 0,C 180,E1 -19498.541,E2 -19498.541} C_VEL
LIN {X 0,Y 248.899,Z 321.097,A -85,B 0,C 180,E1 -19499.63,E2 -19499.63} C_VEL
LIN {X 0,Y 251.609,Z 335.953,A -85,B 0,C 180,E1 -19500.843,E2 -19500.843} C_VEL
LIN {X 0,Y 253.755,Z 354.379,A -85,B 0,C 180,E1 -19502.033,E2 -19502.033} C_VEL
LIN {X 0,Y 253.675,Z 361.387,A -85,B 0,C 180,E1 -19502.325,E2 -19502.325} C_VEL
LIN {X 0,Y 252.249,Z 383.863,A -85,B 0,C 180,E1 -19503.139,E2 -19503.139} C_VEL
LIN {X 0,Y 250.731,Z 396.153,A -85,B 0,C 180,E1 -19503.883,E2 -19503.883} C_VEL
LIN {X 0,Y 249.066,Z 405.844,A -85,B 0,C 180,E1 -19504.73,E2 -19504.73} C_VEL
LIN {X 0,Y 247.327,Z 414.172,A -85,B 0,C 180,E1 -19505.669,E2 -19505.669} C_VEL
LIN {X 0,Y 245.458,Z 422.226,A -85,B 0,C 180,E1 -19506.816,E2 -19506.816} C_VEL
LIN {X 0,Y 243.471,Z 429.961,A -85,B 0,C 180,E1 -19508.184,E2 -19508.184} C_VEL
LIN {X 0,Y 241.108,Z 438.176,A -85,B 0,C 180,E1 -19509.972,E2 -19509.972} C_VEL
LIN {X 0,Y 238.845,Z 445.476,A -85,B 0,C 180,E1 -19512.004,E2 -19512.004} C_VEL
LIN {X 0,Y 237.285,Z 450.256,A -85,B 0,C 180,E1 -19513.658,E2 -19513.658} C_VEL
LIN {X 0,Y 235.432,Z 455.902,A -85,B 0,C 180,E1 -19516.184,E2 -19516.184} C_VEL
LIN {X 0,Y 234.074,Z 460.15,A -85,B 0,C 180,E1 -19518.747,E2 -19518.747} C_VEL
LIN {X 0,Y 233.282,Z 463.15,A -85,B 0,C 180,E1 -19521.337,E2 -19521.337} C_VEL
LIN {X 0,Y 232.979,Z 464.442,A -85,B 0,C 180,E1 -19523.07,E2 -19523.07} C_VEL
LIN {X 0,Y 232.848,Z 465.291,A -85,B 0,C 180,E1 -19524.904,E2 -19524.904} C_VEL
LIN {X 0,Y 232.878,Z 465.624,A -85,B 0,C 180,E1 -19526.54,E2 -19526.54} C_VEL
LIN {X 0,Y 232.959,Z 465.413,A -85,B 0,C 180,E1 -19528.272,E2 -19528.272} C_VEL
LIN {X 0,Y 233.072,Z 464.629,A -85,B 0,C 180,E1 -19530,E2 -19530} C_VEL
LIN {X 0,Y 233.014,Z 463.327,A -85,B 0,C 180,E1 -19531.729,E2 -19531.729} C_VEL
LIN {X 0,Y 233.044,Z 460.34,A -85,B 0,C 180,E1 -19534.324,E2 -19534.324} C_VEL
LIN {X 0,Y 233.137,Z 455.972,A -85,B 0,C 180,E1 -19536.926,E2 -19536.926} C_VEL
LIN {X 0,Y 233.432,Z 451.026,A -85,B 0,C 180,E1 -19539.095,E2 -19539.095} C_VEL
LIN {X 0,Y 233.954,Z 444.715,A -85,B 0,C 180,E1 -19541.26,E2 -19541.26} C_VEL
LIN {X 0,Y 234.608,Z 438.541,A -85,B 0,C 180,E1 -19542.984,E2 -19542.984} C_VEL
LIN {X 0,Y 235.33,Z 432.053,A -85,B 0,C 180,E1 -19544.484,E2 -19544.484} C_VEL
LIN {X 0,Y 236.148,Z 425.464,A -85,B 0,C 180,E1 -19545.758,E2 -19545.758} C_VEL
LIN {X 0,Y 236.915,Z 419.005,A -85,B 0,C 180,E1 -19546.812,E2 -19546.812} C_VEL
LIN {X 0,Y 237.663,Z 411.172,A -85,B 0,C 180,E1 -19547.867,E2 -19547.867} C_VEL
LIN {X 0,Y 238.752,Z 401.255,A -85,B 0,C 180,E1 -19548.893,E2 -19548.893} C_VEL
LIN {X 0,Y 239.46,Z 391.929,A -85,B 0,C 180,E1 -19549.614,E2 -19549.614} C_VEL
LIN {X 0,Y 239.919,Z 382.293,A -85,B 0,C 180,E1 -19550.132,E2 -19550.132} C_VEL
LIN {X 0,Y 240.727,Z 352.035,A -85,B 0,C 180,E1 -19551.218,E2 -19551.218} C_VEL
LIN {X 0,Y 236.465,Z 306.138,A -85,B 0,C 180,E1 -19553.174,E2 -19553.174} C_VEL
LIN {X 0,Y 237.435,Z 299,A -85,B 0,C 180,E1 -19555.887,E2 -19555.887} C_VEL
LIN {X 0,Y 235.833,Z 290.205,A -85,B 0,C 180,E1 -19559.452,E2 -19559.452} C_VEL
LIN {X 0,Y 235.041,Z 286.024,A -85,B 0,C 180,E1 -19561.238,E2 -19561.238} C_VEL
LIN {X 0,Y 234.943,Z 286.03,A -85,B 0,C 180,E1 -19566.13,E2 -19566.13} C_VEL
LIN {X 0,Y 234.945,Z 286.03,A -85,B 0,C 180,E1 -19568.943,E2 -19568.943} C_VEL
LIN {X 0,Y 234.888,Z 286.037,A -85,B 0,C 180,E1 -19573.485,E2 -19573.485} C_VEL
LIN {X 0,Y 234.882,Z 286.037,A -85,B 0,C 180,E1 -19576.511,E2 -19576.511} C_VEL
LIN {X 0,Y 234.919,Z 286.032,A -85,B 0,C 180,E1 -19581.077,E2 -19581.077} C_VEL
LIN {X 0,Y 234.931,Z 286.034,A -85,B 0,C 180,E1 -19585.361,E2 -19585.361} C_VEL
LIN {X 0,Y 234.932,Z 286.033,A -85,B 0,C 180,E1 -19589.431,E2 -19589.431} C_VEL
LIN {X 0,Y 234.995,Z 286.026,A -85,B 0,C 180,E1 -19593.792,E2 -19593.792} C_VEL
LIN {X 0,Y 235.011,Z 286.019,A -85,B 0,C 180,E1 -19598.969,E2 -19598.969} C_VEL
LIN {X 0,Y 235.096,Z 286.012,A -85,B 0,C 180,E1 -19603.058,E2 -19603.058} C_VEL
LIN {X 0,Y 235.112,Z 286.01,A -85,B 0,C 180,E1 -19607.921,E2 -19607.921} C_VEL
LIN {X 0,Y 235.33,Z 285.984,A -85,B 0,C 180,E1 -19611.411,E2 -19611.411} C_VEL
LIN {X 0,Y 235.371,Z 285.977,A -85,B 0,C 180,E1 -19613.139,E2 -19613.139} C_VEL
LIN {X 0,Y 235.593,Z 285.949,A -85,B 0,C 180,E1 -19618.289,E2 -19618.289} C_VEL
LIN {X 0,Y 235.593,Z 285.951,A -85,B 0,C 180,E1 -19621.708,E2 -19621.708} C_VEL
LIN {X 0,Y 235.401,Z 285.973,A -85,B 0,C 180,E1 -19626.857,E2 -19626.857} C_VEL
LIN {X 0,Y 235.235,Z 285.993,A -85,B 0,C 180,E1 -19630.325,E2 -19630.325} C_VEL
LIN {X 0,Y 235.108,Z 286.012,A -85,B 0,C 180,E1 -19635.605,E2 -19635.605} C_VEL
LIN {X 0,Y 235.015,Z 286.021,A -85,B 0,C 180,E1 -19639.203,E2 -19639.203} C_VEL
LIN {X 0,Y 234.976,Z 286.025,A -85,B 0,C 180,E1 -19642.879,E2 -19642.879} C_VEL
LIN {X 0,Y 234.964,Z 286.027,A -85,B 0,C 180,E1 -19646.656,E2 -19646.656} C_VEL
LIN {X 0,Y 234.926,Z 286.03,A -85,B 0,C 180,E1 -19650.566,E2 -19650.566} C_VEL
LIN {X 0,Y 234.955,Z 286.028,A -85,B 0,C 180,E1 -19654.632,E2 -19654.632} C_VEL
LIN {X 0,Y 234.936,Z 286.029,A -85,B 0,C 180,E1 -19658.943,E2 -19658.943} C_VEL
LIN {X 0,Y 234.955,Z 286.031,A -85,B 0,C 180,E1 -19663.468,E2 -19663.468} C_VEL
LIN {X 0,Y 234.959,Z 286.025,A -85,B 0,C 180,E1 -19666.531,E2 -19666.531} C_VEL
LIN {X 0,Y 234.949,Z 286.03,A -85,B 0,C 180,E1 -19671.085,E2 -19671.085} C_VEL
LIN {X 0,Y 234.954,Z 286.027,A -85,B 0,C 180,E1 -19675.366,E2 -19675.366} C_VEL
LIN {X 0,Y 234.963,Z 286.028,A -85,B 0,C 180,E1 -19680.157,E2 -19680.157} C_VEL
LIN {X 0,Y 234.988,Z 286.025,A -85,B 0,C 180,E1 -19683.793,E2 -19683.793} C_VEL
LIN {X 0,Y 235.005,Z 286.022,A -85,B 0,C 180,E1 -19688.969,E2 -19688.969} C_VEL
LIN {X 0,Y 235.09,Z 286.01,A -85,B 0,C 180,E1 -19693.059,E2 -19693.059} C_VEL
LIN {X 0,Y 235.14,Z 286.007,A -85,B 0,C 180,E1 -19697.923,E2 -19697.923} C_VEL
LIN {X 0,Y 235.37,Z 285.976,A -85,B 0,C 180,E1 -19701.414,E2 -19701.414} C_VEL
LIN {X 0,Y 235.396,Z 285.973,A -85,B 0,C 180,E1 -19703.141,E2 -19703.141} C_VEL
LIN {X 0,Y 235.588,Z 285.948,A -85,B 0,C 180,E1 -19708.29,E2 -19708.29} C_VEL
LIN {X 0,Y 235.588,Z 285.952,A -85,B 0,C 180,E1 -19711.709,E2 -19711.709} C_VEL
LIN {X 0,Y 235.394,Z 285.971,A -85,B 0,C 180,E1 -19716.858,E2 -19716.858} C_VEL
LIN {X 0,Y 235.23,Z 285.995,A -85,B 0,C 180,E1 -19720.326,E2 -19720.326} C_VEL
LIN {X 0,Y 235.106,Z 286.01,A -85,B 0,C 180,E1 -19725.606,E2 -19725.606} C_VEL
LIN {X 0,Y 235,Z 286.023,A -85,B 0,C 180,E1 -19729.205,E2 -19729.205} C_VEL
LIN {X 0,Y 234.944,Z 286.03,A -85,B 0,C 180,E1 -19732.884,E2 -19732.884} C_VEL
LIN {X 0,Y 235.015,Z 286.025,A -85,B 0,C 180,E1 -19736.006,E2 -19736.006} C_VEL
LIN {X 0,Y 241.805,Z 306.813,A -85,B 0,C 180,E1 -19737.242,E2 -19737.242} C_VEL
LIN {X 0,Y 240.108,Z 358.14,A -85,B 0,C 180,E1 -19739.064,E2 -19739.064} C_VEL
LIN {X 0,Y 239.648,Z 369.566,A -85,B 0,C 180,E1 -19739.754,E2 -19739.754} C_VEL
LIN {X 0,Y 238.755,Z 381.322,A -85,B 0,C 180,E1 -19740.844,E2 -19740.844} C_VEL
LIN {X 0,Y 238.115,Z 389.559,A -85,B 0,C 180,E1 -19741.854,E2 -19741.854} C_VEL
LIN {X 0,Y 237.311,Z 398.454,A -85,B 0,C 180,E1 -19743.22,E2 -19743.22} C_VEL
LIN {X 0,Y 236.392,Z 406.039,A -85,B 0,C 180,E1 -19744.651,E2 -19744.651} C_VEL
LIN {X 0,Y 235.311,Z 414.735,A -85,B 0,C 180,E1 -19746.678,E2 -19746.678} C_VEL
LIN {X 0,Y 234.514,Z 421.811,A -85,B 0,C 180,E1 -19748.818,E2 -19748.818} C_VEL
LIN {X 0,Y 233.863,Z 426.884,A -85,B 0,C 180,E1 -19750.71,E2 -19750.71} C_VEL
LIN {X 0,Y 233.465,Z 430.929,A -85,B 0,C 180,E1 -19752.559,E2 -19752.559} C_VEL
LIN {X 0,Y 233.011,Z 434.985,A -85,B 0,C 180,E1 -19754.968,E2 -19754.968} C_VEL
LIN {X 0,Y 232.83,Z 436.929,A -85,B 0,C 180,E1 -19756.421,E2 -19756.421} C_VEL
LIN {X 0,Y 232.762,Z 439.265,A -85,B 0,C 180,E1 -19759.01,E2 -19759.01} C_VEL
LIN {X 0,Y 233.037,Z 440.464,A -85,B 0,C 180,E1 -19761.637,E2 -19761.637} C_VEL
LIN {X 0,Y 233.276,Z 440.69,A -85,B 0,C 180,E1 -19762.95,E2 -19762.95} C_VEL
LIN {X 0,Y 233.882,Z 440.29,A -85,B 0,C 180,E1 -19765.187,E2 -19765.187} C_VEL
LIN {X 0,Y 234.751,Z 439.04,A -85,B 0,C 180,E1 -19767.394,E2 -19767.394} C_VEL
LIN {X 0,Y 235.874,Z 436.684,A -85,B 0,C 180,E1 -19769.774,E2 -19769.774} C_VEL
LIN {X 0,Y 237.631,Z 432.528,A -85,B 0,C 180,E1 -19772.528,E2 -19772.528} C_VEL
LIN {X 0,Y 239.836,Z 426.633,A -85,B 0,C 180,E1 -19775.282,E2 -19775.282} C_VEL
LIN {X 0,Y 241.941,Z 420.5,A -85,B 0,C 180,E1 -19777.365,E2 -19777.365} C_VEL
LIN {X 0,Y 243.891,Z 414.12,A -85,B 0,C 180,E1 -19779.11,E2 -19779.11} C_VEL
LIN {X 0,Y 245.82,Z 407.219,A -85,B 0,C 180,E1 -19780.638,E2 -19780.638} C_VEL
LIN {X 0,Y 247.628,Z 399.672,A -85,B 0,C 180,E1 -19782.008,E2 -19782.008} C_VEL
LIN {X 0,Y 249.469,Z 390.805,A -85,B 0,C 180,E1 -19783.298,E2 -19783.298} C_VEL
LIN {X 0,Y 251.268,Z 380.116,A -85,B 0,C 180,E1 -19784.488,E2 -19784.488} C_VEL
LIN {X 0,Y 252.526,Z 369.103,A -85,B 0,C 180,E1 -19785.367,E2 -19785.367} C_VEL
LIN {X 0,Y 253.362,Z 359.316,A -85,B 0,C 180,E1 -19785.897,E2 -19785.897} C_VEL
LIN {X 0,Y 255.431,Z 321.192,A -85,B 0,C 180,E1 -19787.25,E2 -19787.25} C_VEL
LIN {X 0,Y 250.632,Z 311.386,A -85,B 0,C 180,E1 -19788.613,E2 -19788.613} C_VEL
LIN {X 0,Y 244.554,Z 301.138,A -85,B 0,C 180,E1 -19790.369,E2 -19790.369} C_VEL
LIN {X 0,Y 240.343,Z 294.401,A -85,B 0,C 180,E1 -19791.7,E2 -19791.7} C_VEL
LIN {X 0,Y 238.469,Z 291.232,A -85,B 0,C 180,E1 -19792.327,E2 -19792.327} C_VEL
LIN {X 0,Y 236.047,Z 288.267,A -85,B 0,C 180,E1 -19793.108,E2 -19793.108} C_VEL
LIN {X 0,Y 235.363,Z 285.982,A -85,B 0,C 180,E1 -19793.465,E2 -19793.465} C_VEL
LIN {X 0,Y 235.59,Z 285.946,A -85,B 0,C 180,E1 -19798.292,E2 -19798.292} C_VEL
LIN {X 0,Y 235.59,Z 285.945,A -85,B 0,C 180,E1 -19801.711,E2 -19801.711} C_VEL
LIN {X 0,Y 235.399,Z 285.974,A -85,B 0,C 180,E1 -19806.86,E2 -19806.86} C_VEL
LIN {X 0,Y 235.233,Z 285.997,A -85,B 0,C 180,E1 -19810.328,E2 -19810.328} C_VEL
LIN {X 0,Y 235.103,Z 286.005,A -85,B 0,C 180,E1 -19815.608,E2 -19815.608} C_VEL
LIN {X 0,Y 235.004,Z 286.022,A -85,B 0,C 180,E1 -19819.207,E2 -19819.207} C_VEL
LIN {X 0,Y 234.958,Z 286.029,A -85,B 0,C 180,E1 -19822.884,E2 -19822.884} C_VEL
LIN {X 0,Y 234.968,Z 286.024,A -85,B 0,C 180,E1 -19826.659,E2 -19826.659} C_VEL
LIN {X 0,Y 234.967,Z 286.017,A -85,B 0,C 180,E1 -19829.831,E2 -19829.831} C_VEL
LIN {X 0,Y 234.358,Z 286.106,A -85,B 0,C 180,E1 -19831.26,E2 -19831.26} C_VEL
LIN {X 0,Y 231.508,Z 286.452,A -85,B 0,C 180,E1 -19833.589,E2 -19833.589} C_VEL
LIN {X 0,Y 229.037,Z 286.769,A -85,B 0,C 180,E1 -19835.489,E2 -19835.489} C_VEL
LIN {X 0,Y 227.963,Z 286.893,A -85,B 0,C 180,E1 -19836.965,E2 -19836.965} C_VEL
LIN {X 0,Y 227.87,Z 286.904,A -85,B 0,C 180,E1 -19837.466,E2 -19837.466} C_VEL
LIN {X 0,Y 227.886,Z 286.913,A -85,B 0,C 180,E1 -19842.257,E2 -19842.257} C_VEL
LIN {X 0,Y 227.886,Z 287.112,A -85,B 0,C 180,E1 -19846.494,E2 -19846.494} C_VEL
LIN {X 0,Y 230.117,Z 294.307,A -85,B 0,C 180,E1 -19851.151,E2 -19851.151} C_VEL
LIN {X 0,Y 231.791,Z 300.436,A -85,B 0,C 180,E1 -19854.559,E2 -19854.559} C_VEL
LIN {X 0,Y 234.405,Z 305.297,A -85,B 0,C 180,E1 -19855.539,E2 -19855.539} C_VEL
LIN {X 0,Y 238.713,Z 313.403,A -85,B 0,C 180,E1 -19857.039,E2 -19857.039} C_VEL
LIN {X 0,Y 242.827,Z 322.141,A -85,B 0,C 180,E1 -19858.425,E2 -19858.425} C_VEL
LIN {X 0,Y 244.018,Z 325.268,A -85,B 0,C 180,E1 -19858.831,E2 -19858.831} C_VEL
LIN {X 0,Y 246.683,Z 341.502,A -85,B 0,C 180,E1 -19860.15,E2 -19860.15} C_VEL
LIN {X 0,Y 248.204,Z 357.001,A -85,B 0,C 180,E1 -19861.169,E2 -19861.169} C_VEL
LIN {X 0,Y 246.599,Z 382.988,A -85,B 0,C 180,E1 -19862.135,E2 -19862.135} C_VEL
LIN {X 0,Y 245.11,Z 394.876,A -85,B 0,C 180,E1 -19862.839,E2 -19862.839} C_VEL
LIN {X 0,Y 243.481,Z 404.373,A -85,B 0,C 180,E1 -19863.665,E2 -19863.665} C_VEL
LIN {X 0,Y 241.68,Z 412.785,A -85,B 0,C 180,E1 -19864.602,E2 -19864.602} C_VEL
LIN {X 0,Y 239.638,Z 421.019,A -85,B 0,C 180,E1 -19865.759,E2 -19865.759} C_VEL
LIN {X 0,Y 237.52,Z 428.884,A -85,B 0,C 180,E1 -19867.149,E2 -19867.149} C_VEL
LIN {X 0,Y 235.531,Z 435.452,A -85,B 0,C 180,E1 -19868.561,E2 -19868.561} C_VEL
LIN {X 0,Y 233.474,Z 441.75,A -85,B 0,C 180,E1 -19870.206,E2 -19870.206} C_VEL
LIN {X 0,Y 231.678,Z 447.018,A -85,B 0,C 180,E1 -19871.885,E2 -19871.885} C_VEL
LIN {X 0,Y 229.729,Z 452.439,A -85,B 0,C 180,E1 -19874.019,E2 -19874.019} C_VEL
LIN {X 0,Y 228.013,Z 457.559,A -85,B 0,C 180,E1 -19876.635,E2 -19876.635} C_VEL
LIN {X 0,Y 226.785,Z 461.236,A -85,B 0,C 180,E1 -19879.285,E2 -19879.285} C_VEL
LIN {X 0,Y 226.257,Z 463,A -85,B 0,C 180,E1 -19881.066,E2 -19881.066} C_VEL
LIN {X 0,Y 225.92,Z 464.187,A -85,B 0,C 180,E1 -19882.853,E2 -19882.853} C_VEL
LIN {X 0,Y 225.775,Z 464.988,A -85,B 0,C 180,E1 -19884.953,E2 -19884.953} C_VEL
LIN {X 0,Y 225.797,Z 465.172,A -85,B 0,C 180,E1 -19886.432,E2 -19886.432} C_VEL
LIN {X 0,Y 225.886,Z 464.939,A -85,B 0,C 180,E1 -19888.218,E2 -19888.218} C_VEL
LIN {X 0,Y 225.995,Z 464.091,A -85,B 0,C 180,E1 -19890,E2 -19890} C_VEL
LIN {X 0,Y 225.945,Z 462.695,A -85,B 0,C 180,E1 -19891.783,E2 -19891.783} C_VEL
LIN {X 0,Y 226.013,Z 460.766,A -85,B 0,C 180,E1 -19893.566,E2 -19893.566} C_VEL
LIN {X 0,Y 225.953,Z 457.917,A -85,B 0,C 180,E1 -19895.536,E2 -19895.536} C_VEL
LIN {X 0,Y 226.078,Z 455.049,A -85,B 0,C 180,E1 -19897.143,E2 -19897.143} C_VEL
LIN {X 0,Y 226.4,Z 449.939,A -85,B 0,C 180,E1 -19899.38,E2 -19899.38} C_VEL
LIN {X 0,Y 226.806,Z 444.923,A -85,B 0,C 180,E1 -19901.167,E2 -19901.167} C_VEL
LIN {X 0,Y 227.496,Z 438.874,A -85,B 0,C 180,E1 -19902.943,E2 -19902.943} C_VEL
LIN {X 0,Y 228.331,Z 431.494,A -85,B 0,C 180,E1 -19904.711,E2 -19904.711} C_VEL
LIN {X 0,Y 229.148,Z 424.863,A -85,B 0,C 180,E1 -19906.024,E2 -19906.024} C_VEL
LIN {X 0,Y 229.924,Z 418.356,A -85,B 0,C 180,E1 -19907.11,E2 -19907.11} C_VEL
LIN {X 0,Y 230.709,Z 410.468,A -85,B 0,C 180,E1 -19908.194,E2 -19908.194} C_VEL
LIN {X 0,Y 231.707,Z 401.629,A -85,B 0,C 180,E1 -19909.145,E2 -19909.145} C_VEL
LIN {X 0,Y 232.473,Z 392.089,A -85,B 0,C 180,E1 -19909.918,E2 -19909.918} C_VEL
LIN {X 0,Y 232.958,Z 382.336,A -85,B 0,C 180,E1 -19910.47,E2 -19910.47} C_VEL
LIN {X 0,Y 233.81,Z 352.618,A -85,B 0,C 180,E1 -19911.575,E2 -19911.575} C_VEL
LIN {X 0,Y 229.561,Z 305.746,A -85,B 0,C 180,E1 -19913.646,E2 -19913.646} C_VEL
LIN {X 0,Y 230.371,Z 300.325,A -85,B 0,C 180,E1 -19915.768,E2 -19915.768} C_VEL
LIN {X 0,Y 229.609,Z 295.347,A -85,B 0,C 180,E1 -19917.824,E2 -19917.824} C_VEL
LIN {X 0,Y 227.993,Z 286.903,A -85,B 0,C 180,E1 -19921.446,E2 -19921.446} C_VEL
LIN {X 0,Y 227.898,Z 286.907,A -85,B 0,C 180,E1 -19926.696,E2 -19926.696} C_VEL
LIN {X 0,Y 227.837,Z 286.914,A -85,B 0,C 180,E1 -19930.374,E2 -19930.374} C_VEL
LIN {X 0,Y 227.831,Z 286.916,A -85,B 0,C 180,E1 -19935.193,E2 -19935.193} C_VEL
LIN {X 0,Y 227.826,Z 286.918,A -85,B 0,C 180,E1 -19939.622,E2 -19939.622} C_VEL
LIN {X 0,Y 227.882,Z 286.91,A -85,B 0,C 180,E1 -19944.127,E2 -19944.127} C_VEL
LIN {X 0,Y 227.871,Z 286.909,A -85,B 0,C 180,E1 -19948.377,E2 -19948.377} C_VEL
LIN {X 0,Y 227.887,Z 286.908,A -85,B 0,C 180,E1 -19952.444,E2 -19952.444} C_VEL
LIN {X 0,Y 227.914,Z 286.905,A -85,B 0,C 180,E1 -19956.366,E2 -19956.366} C_VEL
LIN {X 0,Y 227.942,Z 286.902,A -85,B 0,C 180,E1 -19960.173,E2 -19960.173} C_VEL
LIN {X 0,Y 228.056,Z 286.889,A -85,B 0,C 180,E1 -19963.896,E2 -19963.896} C_VEL
LIN {X 0,Y 228.07,Z 286.886,A -85,B 0,C 180,E1 -19967.542,E2 -19967.542} C_VEL
LIN {X 0,Y 228.266,Z 286.863,A -85,B 0,C 180,E1 -19971.143,E2 -19971.143} C_VEL
LIN {X 0,Y 228.322,Z 286.855,A -85,B 0,C 180,E1 -19972.926,E2 -19972.926} C_VEL
LIN {X 0,Y 228.552,Z 286.827,A -85,B 0,C 180,E1 -19978.236,E2 -19978.236} C_VEL
LIN {X 0,Y 228.552,Z 286.828,A -85,B 0,C 180,E1 -19981.761,E2 -19981.761} C_VEL
LIN {X 0,Y 228.352,Z 286.851,A -85,B 0,C 180,E1 -19987.07,E2 -19987.07} C_VEL
LIN {X 0,Y 228.156,Z 286.874,A -85,B 0,C 180,E1 -19990.649,E2 -19990.649} C_VEL
LIN {X 0,Y 228.059,Z 286.887,A -85,B 0,C 180,E1 -19994.271,E2 -19994.271} C_VEL
LIN {X 0,Y 228.003,Z 286.896,A -85,B 0,C 180,E1 -19997.952,E2 -19997.952} C_VEL
LIN {X 0,Y 227.956,Z 286.9,A -85,B 0,C 180,E1 -20002.346,E2 -20002.346} C_VEL
LIN {X 0,Y 227.938,Z 286.902,A -85,B 0,C 180,E1 -20006.601,E2 -20006.601} C_VEL
LIN {X 0,Y 227.903,Z 286.906,A -85,B 0,C 180,E1 -20010.294,E2 -20010.294} C_VEL
LIN {X 0,Y 227.885,Z 286.913,A -85,B 0,C 180,E1 -20013.717,E2 -20013.717} C_VEL
LIN {X 0,Y 227.866,Z 286.911,A -85,B 0,C 180,E1 -20018.084,E2 -20018.084} C_VEL
LIN {X 0,Y 227.896,Z 286.908,A -85,B 0,C 180,E1 -20022.72,E2 -20022.72} C_VEL
LIN {X 0,Y 227.903,Z 286.908,A -85,B 0,C 180,E1 -20027.737,E2 -20027.737} C_VEL
LIN {X 0,Y 227.865,Z 286.914,A -85,B 0,C 180,E1 -20031.913,E2 -20031.913} C_VEL
LIN {X 0,Y 227.884,Z 286.909,A -85,B 0,C 180,E1 -20036.372,E2 -20036.372} C_VEL
LIN {X 0,Y 227.913,Z 286.905,A -85,B 0,C 180,E1 -20040.437,E2 -20040.437} C_VEL
LIN {X 0,Y 227.922,Z 286.904,A -85,B 0,C 180,E1 -20044.425,E2 -20044.425} C_VEL
LIN {X 0,Y 227.955,Z 286.901,A -85,B 0,C 180,E1 -20048.286,E2 -20048.286} C_VEL
LIN {X 0,Y 228.028,Z 286.889,A -85,B 0,C 180,E1 -20052.825,E2 -20052.825} C_VEL
LIN {X 0,Y 228.087,Z 286.886,A -85,B 0,C 180,E1 -20057.544,E2 -20057.544} C_VEL
LIN {X 0,Y 228.299,Z 286.855,A -85,B 0,C 180,E1 -20061.146,E2 -20061.146} C_VEL
LIN {X 0,Y 228.347,Z 286.851,A -85,B 0,C 180,E1 -20062.928,E2 -20062.928} C_VEL
LIN {X 0,Y 228.546,Z 286.825,A -85,B 0,C 180,E1 -20068.237,E2 -20068.237} C_VEL
LIN {X 0,Y 228.546,Z 286.83,A -85,B 0,C 180,E1 -20071.762,E2 -20071.762} C_VEL
LIN {X 0,Y 228.345,Z 286.849,A -85,B 0,C 180,E1 -20077.071,E2 -20077.071} C_VEL
LIN {X 0,Y 228.156,Z 286.875,A -85,B 0,C 180,E1 -20080.65,E2 -20080.65} C_VEL
LIN {X 0,Y 228.057,Z 286.887,A -85,B 0,C 180,E1 -20084.272,E2 -20084.272} C_VEL
LIN {X 0,Y 227.995,Z 286.898,A -85,B 0,C 180,E1 -20087.953,E2 -20087.953} C_VEL
LIN {X 0,Y 227.917,Z 286.907,A -85,B 0,C 180,E1 -20092.326,E2 -20092.326} C_VEL
LIN {X 0,Y 227.959,Z 286.909,A -85,B 0,C 180,E1 -20095.57,E2 -20095.57} C_VEL
LIN {X 0,Y 234.846,Z 307.671,A -85,B 0,C 180,E1 -20096.836,E2 -20096.836} C_VEL
LIN {X 0,Y 233.197,Z 358.191,A -85,B 0,C 180,E1 -20098.69,E2 -20098.69} C_VEL
LIN {X 0,Y 232.728,Z 369.644,A -85,B 0,C 180,E1 -20099.394,E2 -20099.394} C_VEL
LIN {X 0,Y 231.815,Z 381.547,A -85,B 0,C 180,E1 -20100.519,E2 -20100.519} C_VEL
LIN {X 0,Y 231.027,Z 390.895,A -85,B 0,C 180,E1 -20101.713,E2 -20101.713} C_VEL
LIN {X 0,Y 230.234,Z 399.604,A -85,B 0,C 180,E1 -20103.117,E2 -20103.117} C_VEL
LIN {X 0,Y 229.075,Z 408.605,A -85,B 0,C 180,E1 -20104.914,E2 -20104.914} C_VEL
LIN {X 0,Y 228.026,Z 416.784,A -85,B 0,C 180,E1 -20107.03,E2 -20107.03} C_VEL
LIN {X 0,Y 227.439,Z 422.126,A -85,B 0,C 180,E1 -20108.718,E2 -20108.718} C_VEL
LIN {X 0,Y 226.779,Z 427.061,A -85,B 0,C 180,E1 -20110.6,E2 -20110.6} C_VEL
LIN {X 0,Y 226.378,Z 431.233,A -85,B 0,C 180,E1 -20112.556,E2 -20112.556} C_VEL
LIN {X 0,Y 226.007,Z 434.349,A -85,B 0,C 180,E1 -20114.342,E2 -20114.342} C_VEL
LIN {X 0,Y 225.696,Z 437.492,A -85,B 0,C 180,E1 -20116.762,E2 -20116.762} C_VEL
LIN {X 0,Y 225.671,Z 439.603,A -85,B 0,C 180,E1 -20119.159,E2 -20119.159} C_VEL
LIN {X 0,Y 225.947,Z 440.77,A -85,B 0,C 180,E1 -20121.533,E2 -20121.533} C_VEL
LIN {X 0,Y 226.382,Z 441.046,A -85,B 0,C 180,E1 -20123.856,E2 -20123.856} C_VEL
LIN {X 0,Y 227.29,Z 440.244,A -85,B 0,C 180,E1 -20126.599,E2 -20126.599} C_VEL
LIN {X 0,Y 228.572,Z 438.169,A -85,B 0,C 180,E1 -20129.418,E2 -20129.418} C_VEL
LIN {X 0,Y 230.315,Z 434.588,A -85,B 0,C 180,E1 -20132.239,E2 -20132.239} C_VEL
LIN {X 0,Y 231.982,Z 430.65,A -85,B 0,C 180,E1 -20134.426,E2 -20134.426} C_VEL
LIN {X 0,Y 233.927,Z 425.612,A -85,B 0,C 180,E1 -20136.572,E2 -20136.572} C_VEL
LIN {X 0,Y 235.998,Z 419.905,A -85,B 0,C 180,E1 -20138.483,E2 -20138.483} C_VEL
LIN {X 0,Y 238.17,Z 412.998,A -85,B 0,C 180,E1 -20140.344,E2 -20140.344} C_VEL
LIN {X 0,Y 240.602,Z 404.562,A -85,B 0,C 180,E1 -20142.141,E2 -20142.141} C_VEL
LIN {X 0,Y 242.648,Z 395.796,A -85,B 0,C 180,E1 -20143.598,E2 -20143.598} C_VEL
LIN {X 0,Y 244.636,Z 385.494,A -85,B 0,C 180,E1 -20144.911,E2 -20144.911} C_VEL
LIN {X 0,Y 246.072,Z 376.363,A -85,B 0,C 180,E1 -20145.798,E2 -20145.798} C_VEL
LIN {X 0,Y 247.297,Z 365.461,A -85,B 0,C 180,E1 -20146.595,E2 -20146.595} C_VEL
LIN {X 0,Y 248.25,Z 350.681,A -85,B 0,C 180,E1 -20147.238,E2 -20147.238} C_VEL
LIN {X 0,Y 249.825,Z 323.466,A -85,B 0,C 180,E1 -20148.202,E2 -20148.202} C_VEL
LIN {X 0,Y 244.405,Z 312.855,A -85,B 0,C 180,E1 -20149.82,E2 -20149.82} C_VEL
LIN {X 0,Y 238.502,Z 302.969,A -85,B 0,C 180,E1 -20151.689,E2 -20151.689} C_VEL
LIN {X 0,Y 233.918,Z 295.807,A -85,B 0,C 180,E1 -20153.245,E2 -20153.245} C_VEL
LIN {X 0,Y 231.792,Z 292.576,A -85,B 0,C 180,E1 -20154.018,E2 -20154.018} C_VEL
LIN {X 0,Y 231.072,Z 291.725,A -85,B 0,C 180,E1 -20154.273,E2 -20154.273} C_VEL
LIN {X 0,Y 229.053,Z 289.503,A -85,B 0,C 180,E1 -20154.996,E2 -20154.996} C_VEL
LIN {X 0,Y 228.192,Z 286.869,A -85,B 0,C 180,E1 -20155.475,E2 -20155.475} C_VEL
LIN {X 0,Y 228.549,Z 286.822,A -85,B 0,C 180,E1 -20158.239,E2 -20158.239} C_VEL
LIN {X 0,Y 228.549,Z 286.822,A -85,B 0,C 180,E1 -20161.764,E2 -20161.764} C_VEL
LIN {X 0,Y 228.35,Z 286.85,A -85,B 0,C 180,E1 -20167.073,E2 -20167.073} C_VEL
LIN {X 0,Y 228.154,Z 286.877,A -85,B 0,C 180,E1 -20170.652,E2 -20170.652} C_VEL
LIN {X 0,Y 228.055,Z 286.889,A -85,B 0,C 180,E1 -20174.274,E2 -20174.274} C_VEL
LIN {X 0,Y 227.999,Z 286.89,A -85,B 0,C 180,E1 -20177.955,E2 -20177.955} C_VEL
LIN {X 0,Y 227.927,Z 286.899,A -85,B 0,C 180,E1 -20182.331,E2 -20182.331} C_VEL
LIN {X 0,Y 227.941,Z 286.898,A -85,B 0,C 180,E1 -20186.605,E2 -20186.605} C_VEL
LIN {X 0,Y 227.907,Z 286.899,A -85,B 0,C 180,E1 -20190.298,E2 -20190.298} C_VEL
LIN {X 0,Y 227.888,Z 286.9,A -85,B 0,C 180,E1 -20193.72,E2 -20193.72} C_VEL
LIN {X 0,Y 227.87,Z 286.904,A -85,B 0,C 180,E1 -20197.466,E2 -20197.466} C_VEL
LIN {X 0,Y 227.18,Z 286.997,A -85,B 0,C 180,E1 -20198.448,E2 -20198.448} C_VEL
LIN {X 0,Y 224.337,Z 287.35,A -85,B 0,C 180,E1 -20199.99,E2 -20199.99} C_VEL
LIN {X 0,Y 221.485,Z 287.706,A -85,B 0,C 180,E1 -20201.571,E2 -20201.571} C_VEL
LIN {X 0,Y 220.824,Z 287.787,A -85,B 0,C 180,E1 -20202.595,E2 -20202.595} C_VEL
LIN {X 0,Y 220.826,Z 287.998,A -85,B 0,C 180,E1 -20204.442,E2 -20204.442} C_VEL
LIN {X 0,Y 222.878,Z 294.593,A -85,B 0,C 180,E1 -20209.184,E2 -20209.184} C_VEL
LIN {X 0,Y 224.442,Z 299.709,A -85,B 0,C 180,E1 -20212.341,E2 -20212.341} C_VEL
LIN {X 0,Y 227.353,Z 304.776,A -85,B 0,C 180,E1 -20213.553,E2 -20213.553} C_VEL
LIN {X 0,Y 231.506,Z 312.361,A -85,B 0,C 180,E1 -20215.177,E2 -20215.177} C_VEL
LIN {X 0,Y 235.693,Z 320.513,A -85,B 0,C 180,E1 -20216.69,E2 -20216.69} C_VEL
LIN {X 0,Y 238.961,Z 328.198,A -85,B 0,C 180,E1 -20217.872,E2 -20217.872} C_VEL
LIN {X 0,Y 241.389,Z 343.995,A -85,B 0,C 180,E1 -20219.194,E2 -20219.194} C_VEL
LIN {X 0,Y 242.706,Z 358.189,A -85,B 0,C 180,E1 -20220.153,E2 -20220.153} C_VEL
LIN {X 0,Y 241.066,Z 382.514,A -85,B 0,C 180,E1 -20221.079,E2 -20221.079} C_VEL
LIN {X 0,Y 239.353,Z 395.191,A -85,B 0,C 180,E1 -20221.861,E2 -20221.861} C_VEL
LIN {X 0,Y 237.586,Z 404.792,A -85,B 0,C 180,E1 -20222.731,E2 -20222.731} C_VEL
LIN {X 0,Y 235.734,Z 412.933,A -85,B 0,C 180,E1 -20223.675,E2 -20223.675} C_VEL
LIN {X 0,Y 233.592,Z 421.031,A -85,B 0,C 180,E1 -20224.852,E2 -20224.852} C_VEL
LIN {X 0,Y 231.362,Z 428.831,A -85,B 0,C 180,E1 -20226.267,E2 -20226.267} C_VEL
LIN {X 0,Y 228.986,Z 436.205,A -85,B 0,C 180,E1 -20227.916,E2 -20227.916} C_VEL
LIN {X 0,Y 226.403,Z 443.747,A -85,B 0,C 180,E1 -20230.035,E2 -20230.035} C_VEL
LIN {X 0,Y 223.673,Z 450.712,A -85,B 0,C 180,E1 -20232.633,E2 -20232.633} C_VEL
LIN {X 0,Y 221.636,Z 456.066,A -85,B 0,C 180,E1 -20235.306,E2 -20235.306} C_VEL
LIN {X 0,Y 220.145,Z 460.066,A -85,B 0,C 180,E1 -20238.024,E2 -20238.024} C_VEL
LIN {X 0,Y 219.223,Z 462.811,A -85,B 0,C 180,E1 -20240.777,E2 -20240.777} C_VEL
LIN {X 0,Y 218.856,Z 463.936,A -85,B 0,C 180,E1 -20242.621,E2 -20242.621} C_VEL
LIN {X 0,Y 218.697,Z 464.693,A -85,B 0,C 180,E1 -20245.021,E2 -20245.021} C_VEL
LIN {X 0,Y 218.814,Z 464.408,A -85,B 0,C 180,E1 -20248.16,E2 -20248.16} C_VEL
LIN {X 0,Y 218.92,Z 463.534,A -85,B 0,C 180,E1 -20250,E2 -20250} C_VEL
LIN {X 0,Y 218.894,Z 461.152,A -85,B 0,C 180,E1 -20252.761,E2 -20252.761} C_VEL
LIN {X 0,Y 218.89,Z 457.366,A -85,B 0,C 180,E1 -20255.528,E2 -20255.528} C_VEL
LIN {X 0,Y 219.117,Z 452.125,A -85,B 0,C 180,E1 -20258.299,E2 -20258.299} C_VEL
LIN {X 0,Y 219.575,Z 446.446,A -85,B 0,C 180,E1 -20260.606,E2 -20260.606} C_VEL
LIN {X 0,Y 220.366,Z 439.201,A -85,B 0,C 180,E1 -20262.9,E2 -20262.9} C_VEL
LIN {X 0,Y 221.19,Z 431.96,A -85,B 0,C 180,E1 -20264.726,E2 -20264.726} C_VEL
LIN {X 0,Y 222.175,Z 424.268,A -85,B 0,C 180,E1 -20266.305,E2 -20266.305} C_VEL
LIN {X 0,Y 222.936,Z 417.706,A -85,B 0,C 180,E1 -20267.427,E2 -20267.427} C_VEL
LIN {X 0,Y 223.763,Z 409.765,A -85,B 0,C 180,E1 -20268.543,E2 -20268.543} C_VEL
LIN {X 0,Y 224.788,Z 400.847,A -85,B 0,C 180,E1 -20269.521,E2 -20269.521} C_VEL
LIN {X 0,Y 225.55,Z 391.356,A -85,B 0,C 180,E1 -20270.305,E2 -20270.305} C_VEL
LIN {X 0,Y 226.062,Z 381.589,A -85,B 0,C 180,E1 -20270.866,E2 -20270.866} C_VEL
LIN {X 0,Y 226.919,Z 353.402,A -85,B 0,C 180,E1 -20271.945,E2 -20271.945} C_VEL
LIN {X 0,Y 222.663,Z 305.409,A -85,B 0,C 180,E1 -20274.129,E2 -20274.129} C_VEL
LIN {X 0,Y 223.321,Z 300.431,A -85,B 0,C 180,E1 -20276.141,E2 -20276.141} C_VEL
LIN {X 0,Y 221.657,Z 291.591,A -85,B 0,C 180,E1 -20279.959,E2 -20279.959} C_VEL
LIN {X 0,Y 220.928,Z 287.781,A -85,B 0,C 180,E1 -20281.752,E2 -20281.752} C_VEL
LIN {X 0,Y 220.842,Z 287.788,A -85,B 0,C 180,E1 -20287.287,E2 -20287.287} C_VEL
LIN {X 0,Y 220.778,Z 287.793,A -85,B 0,C 180,E1 -20291.95,E2 -20291.95} C_VEL
LIN {X 0,Y 220.772,Z 287.798,A -85,B 0,C 180,E1 -20295.544,E2 -20295.544} C_VEL
LIN {X 0,Y 220.808,Z 287.788,A -85,B 0,C 180,E1 -20300.462,E2 -20300.462} C_VEL
LIN {X 0,Y 220.803,Z 287.792,A -85,B 0,C 180,E1 -20305.044,E2 -20305.044} C_VEL
LIN {X 0,Y 220.869,Z 287.784,A -85,B 0,C 180,E1 -20309.394,E2 -20309.394} C_VEL
LIN {X 0,Y 220.896,Z 287.783,A -85,B 0,C 180,E1 -20313.548,E2 -20313.548} C_VEL
LIN {X 0,Y 220.878,Z 287.783,A -85,B 0,C 180,E1 -20317.552,E2 -20317.552} C_VEL
LIN {X 0,Y 220.984,Z 287.769,A -85,B 0,C 180,E1 -20322.57,E2 -20322.57} C_VEL
LIN {X 0,Y 221.009,Z 287.763,A -85,B 0,C 180,E1 -20327.137,E2 -20327.137} C_VEL
LIN {X 0,Y 221.203,Z 287.742,A -85,B 0,C 180,E1 -20330.858,E2 -20330.858} C_VEL
LIN {X 0,Y 221.257,Z 287.734,A -85,B 0,C 180,E1 -20332.699,E2 -20332.699} C_VEL
LIN {X 0,Y 221.51,Z 287.704,A -85,B 0,C 180,E1 -20338.18,E2 -20338.18} C_VEL
LIN {X 0,Y 221.51,Z 287.704,A -85,B 0,C 180,E1 -20341.817,E2 -20341.817} C_VEL
LIN {X 0,Y 221.303,Z 287.73,A -85,B 0,C 180,E1 -20347.296,E2 -20347.296} C_VEL
LIN {X 0,Y 221.103,Z 287.753,A -85,B 0,C 180,E1 -20350.993,E2 -20350.993} C_VEL
LIN {X 0,Y 221.013,Z 287.765,A -85,B 0,C 180,E1 -20356.628,E2 -20356.628} C_VEL
LIN {X 0,Y 220.905,Z 287.775,A -85,B 0,C 180,E1 -20360.483,E2 -20360.483} C_VEL
LIN {X 0,Y 220.868,Z 287.783,A -85,B 0,C 180,E1 -20364.433,E2 -20364.433} C_VEL
LIN {X 0,Y 220.831,Z 287.785,A -85,B 0,C 180,E1 -20368.512,E2 -20368.512} C_VEL
LIN {X 0,Y 220.819,Z 287.789,A -85,B 0,C 180,E1 -20372.753,E2 -20372.753} C_VEL
LIN {X 0,Y 220.833,Z 287.787,A -85,B 0,C 180,E1 -20377.287,E2 -20377.287} C_VEL
LIN {X 0,Y 220.835,Z 287.79,A -85,B 0,C 180,E1 -20381.935,E2 -20381.935} C_VEL
LIN {X 0,Y 220.862,Z 287.781,A -85,B 0,C 180,E1 -20387.041,E2 -20387.041} C_VEL
LIN {X 0,Y 220.85,Z 287.786,A -85,B 0,C 180,E1 -20390.473,E2 -20390.473} C_VEL
LIN {X 0,Y 220.809,Z 287.787,A -85,B 0,C 180,E1 -20395.047,E2 -20395.047} C_VEL
LIN {X 0,Y 220.862,Z 287.786,A -85,B 0,C 180,E1 -20399.394,E2 -20399.394} C_VEL
LIN {X 0,Y 220.889,Z 287.78,A -85,B 0,C 180,E1 -20403.549,E2 -20403.549} C_VEL
LIN {X 0,Y 220.871,Z 287.785,A -85,B 0,C 180,E1 -20407.553,E2 -20407.553} C_VEL
LIN {X 0,Y 220.978,Z 287.768,A -85,B 0,C 180,E1 -20412.571,E2 -20412.571} C_VEL
LIN {X 0,Y 221.019,Z 287.765,A -85,B 0,C 180,E1 -20417.139,E2 -20417.139} C_VEL
LIN {X 0,Y 221.229,Z 287.735,A -85,B 0,C 180,E1 -20420.86,E2 -20420.86} C_VEL
LIN {X 0,Y 221.283,Z 287.731,A -85,B 0,C 180,E1 -20422.701,E2 -20422.701} C_VEL
LIN {X 0,Y 221.504,Z 287.702,A -85,B 0,C 180,E1 -20428.181,E2 -20428.181} C_VEL
LIN {X 0,Y 221.504,Z 287.707,A -85,B 0,C 180,E1 -20431.818,E2 -20431.818} C_VEL
LIN {X 0,Y 221.281,Z 287.73,A -85,B 0,C 180,E1 -20437.298,E2 -20437.298} C_VEL
LIN {X 0,Y 221.105,Z 287.754,A -85,B 0,C 180,E1 -20440.994,E2 -20440.994} C_VEL
LIN {X 0,Y 221.009,Z 287.766,A -85,B 0,C 180,E1 -20446.63,E2 -20446.63} C_VEL
LIN {X 0,Y 220.877,Z 287.783,A -85,B 0,C 180,E1 -20450.487,E2 -20450.487} C_VEL
LIN {X 0,Y 220.923,Z 287.777,A -85,B 0,C 180,E1 -20455.055,E2 -20455.055} C_VEL
LIN {X 0,Y 228.006,Z 309.301,A -85,B 0,C 180,E1 -20456.447,E2 -20456.447} C_VEL
LIN {X 0,Y 226.257,Z 359.02,A -85,B 0,C 180,E1 -20458.337,E2 -20458.337} C_VEL
LIN {X 0,Y 225.708,Z 370.932,A -85,B 0,C 180,E1 -20459.111,E2 -20459.111} C_VEL
LIN {X 0,Y 224.81,Z 382.473,A -85,B 0,C 180,E1 -20460.27,E2 -20460.27} C_VEL
LIN {X 0,Y 224.033,Z 391.263,A -85,B 0,C 180,E1 -20461.434,E2 -20461.434} C_VEL
LIN {X 0,Y 223.199,Z 400.06,A -85,B 0,C 180,E1 -20462.898,E2 -20462.898} C_VEL
LIN {X 0,Y 222.01,Z 408.97,A -85,B 0,C 180,E1 -20464.736,E2 -20464.736} C_VEL
LIN {X 0,Y 221.106,Z 416.055,A -85,B 0,C 180,E1 -20466.581,E2 -20466.581} C_VEL
LIN {X 0,Y 220.105,Z 423.646,A -85,B 0,C 180,E1 -20469.094,E2 -20469.094} C_VEL
LIN {X 0,Y 219.598,Z 428.342,A -85,B 0,C 180,E1 -20471.024,E2 -20471.024} C_VEL
LIN {X 0,Y 219.148,Z 432.53,A -85,B 0,C 180,E1 -20473.152,E2 -20473.152} C_VEL
LIN {X 0,Y 218.653,Z 437.159,A -85,B 0,C 180,E1 -20476.289,E2 -20476.289} C_VEL
LIN {X 0,Y 218.567,Z 438.579,A -85,B 0,C 180,E1 -20477.692,E2 -20477.692} C_VEL
LIN {X 0,Y 218.687,Z 440.616,A -85,B 0,C 180,E1 -20480.468,E2 -20480.468} C_VEL
LIN {X 0,Y 219.162,Z 441.514,A -85,B 0,C 180,E1 -20483.29,E2 -20483.29} C_VEL
LIN {X 0,Y 220.028,Z 441.134,A -85,B 0,C 180,E1 -20486.145,E2 -20486.145} C_VEL
LIN {X 0,Y 221.505,Z 439.059,A -85,B 0,C 180,E1 -20489.494,E2 -20489.494} C_VEL
LIN {X 0,Y 222.996,Z 436.413,A -85,B 0,C 180,E1 -20491.937,E2 -20491.937} C_VEL
LIN {X 0,Y 225.182,Z 431.841,A -85,B 0,C 180,E1 -20494.833,E2 -20494.833} C_VEL
LIN {X 0,Y 227.214,Z 426.973,A -85,B 0,C 180,E1 -20497.042,E2 -20497.042} C_VEL
LIN {X 0,Y 229.23,Z 421.839,A -85,B 0,C 180,E1 -20498.887,E2 -20498.887} C_VEL
LIN {X 0,Y 231.727,Z 414.46,A -85,B 0,C 180,E1 -20500.988,E2 -20500.988} C_VEL
LIN {X 0,Y 233.842,Z 407.764,A -85,B 0,C 180,E1 -20502.511,E2 -20502.511} C_VEL
LIN {X 0,Y 236.082,Z 399.245,A -85,B 0,C 180,E1 -20504.102,E2 -20504.102} C_VEL
LIN {X 0,Y 238.556,Z 388.149,A -85,B 0,C 180,E1 -20505.665,E2 -20505.665} C_VEL
LIN {X 0,Y 240.08,Z 379.551,A -85,B 0,C 180,E1 -20506.575,E2 -20506.575} C_VEL
LIN {X 0,Y 241.325,Z 369.747,A -85,B 0,C 180,E1 -20507.376,E2 -20507.376} C_VEL
LIN {X 0,Y 242.219,Z 359.887,A -85,B 0,C 180,E1 -20507.934,E2 -20507.934} C_VEL
LIN {X 0,Y 244.323,Z 325.921,A -85,B 0,C 180,E1 -20509.194,E2 -20509.194} C_VEL
LIN {X 0,Y 239.059,Z 315.664,A -85,B 0,C 180,E1 -20510.883,E2 -20510.883} C_VEL
LIN {X 0,Y 232.498,Z 304.752,A -85,B 0,C 180,E1 -20513.111,E2 -20513.111} C_VEL
LIN {X 0,Y 230.148,Z 301.14,A -85,B 0,C 180,E1 -20513.976,E2 -20513.976} C_VEL
LIN {X 0,Y 227.54,Z 297.386,A -85,B 0,C 180,E1 -20514.963,E2 -20514.963} C_VEL
LIN {X 0,Y 225.316,Z 294.532,A -85,B 0,C 180,E1 -20515.827,E2 -20515.827} C_VEL
LIN {X 0,Y 224.522,Z 292.91,A -85,B 0,C 180,E1 -20516.188,E2 -20516.188} C_VEL
LIN {X 0,Y 222.355,Z 290.693,A -85,B 0,C 180,E1 -20517.057,E2 -20517.057} C_VEL
LIN {X 0,Y 221.426,Z 288.149,A -85,B 0,C 180,E1 -20517.557,E2 -20517.557} C_VEL
LIN {X 0,Y 221.389,Z 287.713,A -85,B 0,C 180,E1 -20517.614,E2 -20517.614} C_VEL
LIN {X 0,Y 221.579,Z 287.693,A -85,B 0,C 180,E1 -20520.002,E2 -20520.002} C_VEL
LIN {X 0,Y 221.507,Z 287.7,A -85,B 0,C 180,E1 -20521.82,E2 -20521.82} C_VEL
LIN {X 0,Y 221.285,Z 287.727,A -85,B 0,C 180,E1 -20527.3,E2 -20527.3} C_VEL
LIN {X 0,Y 221.102,Z 287.753,A -85,B 0,C 180,E1 -20530.996,E2 -20530.996} C_VEL
LIN {X 0,Y 221.011,Z 287.754,A -85,B 0,C 180,E1 -20536.632,E2 -20536.632} C_VEL
LIN {X 0,Y 220.889,Z 287.769,A -85,B 0,C 180,E1 -20540.488,E2 -20540.488} C_VEL
LIN {X 0,Y 220.865,Z 287.774,A -85,B 0,C 180,E1 -20544.437,E2 -20544.437} C_VEL
LIN {X 0,Y 220.836,Z 287.78,A -85,B 0,C 180,E1 -20548.515,E2 -20548.515} C_VEL
LIN {X 0,Y 220.823,Z 287.782,A -85,B 0,C 180,E1 -20552.757,E2 -20552.757} C_VEL
LIN {X 0,Y 220.826,Z 287.78,A -85,B 0,C 180,E1 -20557.43,E2 -20557.43} C_VEL
LIN {X 0,Y 220.829,Z 287.789,A -85,B 0,C 180,E1 -20561.94,E2 -20561.94} C_VEL
LIN {X 0,Y 220.824,Z 287.787,A -85,B 0,C 180,E1 -20562.595,E2 -20562.595} C_VEL
LIN {X 0,Y 220.296,Z 288.355,A -85,B 0,C 180,E1 -20563.597,E2 -20563.597} C_VEL
LIN {X 0,Y 218.609,Z 290.294,A -85,B 0,C 180,E1 -20564.826,E2 -20564.826} C_VEL
LIN {X 0,Y 216.145,Z 294.15,A -85,B 0,C 180,E1 -20566.628,E2 -20566.628} C_VEL
LIN {X 0,Y 215.96,Z 295.822,A -85,B 0,C 180,E1 -20567.61,E2 -20567.61} C_VEL
LIN {X 0,Y 217.014,Z 298.979,A -85,B 0,C 180,E1 -20569.718,E2 -20569.718} C_VEL
LIN {X 0,Y 219.823,Z 303.721,A -85,B 0,C 180,E1 -20571.077,E2 -20571.077} C_VEL
LIN {X 0,Y 221.291,Z 305.941,A -85,B 0,C 180,E1 -20571.728,E2 -20571.728} C_VEL
LIN {X 0,Y 224.753,Z 312.059,A -85,B 0,C 180,E1 -20573.225,E2 -20573.225} C_VEL
LIN {X 0,Y 227.994,Z 318.233,A -85,B 0,C 180,E1 -20574.552,E2 -20574.552} C_VEL
LIN {X 0,Y 231.674,Z 325.766,A -85,B 0,C 180,E1 -20575.976,E2 -20575.976} C_VEL
LIN {X 0,Y 234.078,Z 331.428,A -85,B 0,C 180,E1 -20576.885,E2 -20576.885} C_VEL
LIN {X 0,Y 236.205,Z 346.569,A -85,B 0,C 180,E1 -20578.198,E2 -20578.198} C_VEL
LIN {X 0,Y 237.273,Z 359.889,A -85,B 0,C 180,E1 -20579.12,E2 -20579.12} C_VEL
LIN {X 0,Y 235.666,Z 381.996,A -85,B 0,C 180,E1 -20579.972,E2 -20579.972} C_VEL
LIN {X 0,Y 233.829,Z 394.821,A -85,B 0,C 180,E1 -20580.765,E2 -20580.765} C_VEL
LIN {X 0,Y 232.057,Z 404.091,A -85,B 0,C 180,E1 -20581.614,E2 -20581.614} C_VEL
LIN {X 0,Y 230.209,Z 411.844,A -85,B 0,C 180,E1 -20582.507,E2 -20582.507} C_VEL
LIN {X 0,Y 227.967,Z 420.026,A -85,B 0,C 180,E1 -20583.695,E2 -20583.695} C_VEL
LIN {X 0,Y 225.589,Z 427.878,A -85,B 0,C 180,E1 -20585.13,E2 -20585.13} C_VEL
LIN {X 0,Y 223.081,Z 435.294,A -85,B 0,C 180,E1 -20586.81,E2 -20586.81} C_VEL
LIN {X 0,Y 220.241,Z 442.893,A -85,B 0,C 180,E1 -20588.963,E2 -20588.963} C_VEL
LIN {X 0,Y 217.813,Z 448.977,A -85,B 0,C 180,E1 -20591.177,E2 -20591.177} C_VEL
LIN {X 0,Y 216.113,Z 452.946,A -85,B 0,C 180,E1 -20592.982,E2 -20592.982} C_VEL
LIN {X 0,Y 214.2,Z 457.621,A -85,B 0,C 180,E1 -20595.755,E2 -20595.755} C_VEL
LIN {X 0,Y 212.799,Z 460.96,A -85,B 0,C 180,E1 -20598.571,E2 -20598.571} C_VEL
LIN {X 0,Y 212.185,Z 462.584,A -85,B 0,C 180,E1 -20600.468,E2 -20600.468} C_VEL
LIN {X 0,Y 211.816,Z 463.683,A -85,B 0,C 180,E1 -20602.374,E2 -20602.374} C_VEL
LIN {X 0,Y 211.61,Z 464.355,A -85,B 0,C 180,E1 -20605.124,E2 -20605.124} C_VEL
LIN {X 0,Y 211.744,Z 463.849,A -85,B 0,C 180,E1 -20608.098,E2 -20608.098} C_VEL
LIN {X 0,Y 211.847,Z 462.934,A -85,B 0,C 180,E1 -20610,E2 -20610} C_VEL
LIN {X 0,Y 211.837,Z 460.377,A -85,B 0,C 180,E1 -20612.853,E2 -20612.853} C_VEL
LIN {X 0,Y 211.811,Z 456.842,A -85,B 0,C 180,E1 -20615.479,E2 -20615.479} C_VEL
LIN {X 0,Y 211.964,Z 453.039,A -85,B 0,C 180,E1 -20617.622,E2 -20617.622} C_VEL
LIN {X 0,Y 212.355,Z 447.661,A -85,B 0,C 180,E1 -20620.006,E2 -20620.006} C_VEL
LIN {X 0,Y 212.878,Z 442.352,A -85,B 0,C 180,E1 -20621.908,E2 -20621.908} C_VEL
LIN {X 0,Y 213.617,Z 435.951,A -85,B 0,C 180,E1 -20623.8,E2 -20623.8} C_VEL
LIN {X 0,Y 214.788,Z 427.142,A -85,B 0,C 180,E1 -20625.905,E2 -20625.905} C_VEL
LIN {X 0,Y 215.861,Z 418.394,A -85,B 0,C 180,E1 -20627.527,E2 -20627.527} C_VEL
LIN {X 0,Y 216.834,Z 408.862,A -85,B 0,C 180,E1 -20628.912,E2 -20628.912} C_VEL
LIN {X 0,Y 217.9,Z 399.846,A -85,B 0,C 180,E1 -20629.918,E2 -20629.918} C_VEL
LIN {X 0,Y 218.665,Z 390.006,A -85,B 0,C 180,E1 -20630.741,E2 -20630.741} C_VEL
LIN {X 0,Y 219.282,Z 378.702,A -85,B 0,C 180,E1 -20631.371,E2 -20631.371} C_VEL
LIN {X 0,Y 219.981,Z 353.855,A -85,B 0,C 180,E1 -20632.337,E2 -20632.337} C_VEL
LIN {X 0,Y 215.716,Z 304.94,A -85,B 0,C 180,E1 -20634.669,E2 -20634.669} C_VEL
LIN {X 0,Y 216.252,Z 301.696,A -85,B 0,C 180,E1 -20636.023,E2 -20636.023} C_VEL
LIN {X 0,Y 215.269,Z 295.638,A -85,B 0,C 180,E1 -20638.701,E2 -20638.701} C_VEL
LIN {X 0,Y 213.865,Z 288.66,A -85,B 0,C 180,E1 -20641.929,E2 -20641.929} C_VEL
LIN {X 0,Y 213.747,Z 288.669,A -85,B 0,C 180,E1 -20646.287,E2 -20646.287} C_VEL
LIN {X 0,Y 213.72,Z 288.674,A -85,B 0,C 180,E1 -20651.123,E2 -20651.123} C_VEL
LIN {X 0,Y 213.709,Z 288.676,A -85,B 0,C 180,E1 -20653.677,E2 -20653.677} C_VEL
LIN {X 0,Y 213.705,Z 288.676,A -85,B 0,C 180,E1 -20656.344,E2 -20656.344} C_VEL
LIN {X 0,Y 213.718,Z 288.675,A -85,B 0,C 180,E1 -20659.142,E2 -20659.142} C_VEL
LIN {X 0,Y 213.745,Z 288.673,A -85,B 0,C 180,E1 -20663.71,E2 -20663.71} C_VEL
LIN {X 0,Y 213.782,Z 288.664,A -85,B 0,C 180,E1 -20668.73,E2 -20668.73} C_VEL
LIN {X 0,Y 213.827,Z 288.66,A -85,B 0,C 180,E1 -20672.602,E2 -20672.602} C_VEL
LIN {X 0,Y 213.853,Z 288.656,A -85,B 0,C 180,E1 -20676.952,E2 -20676.952} C_VEL
LIN {X 0,Y 213.943,Z 288.646,A -85,B 0,C 180,E1 -20682.802,E2 -20682.802} C_VEL
LIN {X 0,Y 213.951,Z 288.641,A -85,B 0,C 180,E1 -20686.705,E2 -20686.705} C_VEL
LIN {X 0,Y 214.141,Z 288.621,A -85,B 0,C 180,E1 -20690.554,E2 -20690.554} C_VEL
LIN {X 0,Y 214.099,Z 288.624,A -85,B 0,C 180,E1 -20694.347,E2 -20694.347} C_VEL
LIN {X 0,Y 214.443,Z 288.585,A -85,B 0,C 180,E1 -20698.12,E2 -20698.12} C_VEL
LIN {X 0,Y 214.548,Z 288.572,A -85,B 0,C 180,E1 -20699.998,E2 -20699.998} C_VEL
LIN {X 0,Y 214.443,Z 288.584,A -85,B 0,C 180,E1 -20701.876,E2 -20701.876} C_VEL
LIN {X 0,Y 214.237,Z 288.612,A -85,B 0,C 180,E1 -20707.538,E2 -20707.538} C_VEL
LIN {X 0,Y 214.02,Z 288.637,A -85,B 0,C 180,E1 -20711.361,E2 -20711.361} C_VEL
LIN {X 0,Y 213.929,Z 288.648,A -85,B 0,C 180,E1 -20715.235,E2 -20715.235} C_VEL
LIN {X 0,Y 213.872,Z 288.655,A -85,B 0,C 180,E1 -20719.182,E2 -20719.182} C_VEL
LIN {X 0,Y 213.852,Z 288.657,A -85,B 0,C 180,E1 -20723.225,E2 -20723.225} C_VEL
LIN {X 0,Y 213.825,Z 288.662,A -85,B 0,C 180,E1 -20727.448,E2 -20727.448} C_VEL
LIN {X 0,Y 213.775,Z 288.669,A -85,B 0,C 180,E1 -20731.734,E2 -20731.734} C_VEL
LIN {X 0,Y 213.749,Z 288.669,A -85,B 0,C 180,E1 -20736.285,E2 -20736.285} C_VEL
LIN {X 0,Y 213.76,Z 288.668,A -85,B 0,C 180,E1 -20740.871,E2 -20740.871} C_VEL
LIN {X 0,Y 213.803,Z 288.666,A -85,B 0,C 180,E1 -20743.684,E2 -20743.684} C_VEL
LIN {X 0,Y 213.806,Z 288.66,A -85,B 0,C 180,E1 -20746.347,E2 -20746.347} C_VEL
LIN {X 0,Y 213.789,Z 288.665,A -85,B 0,C 180,E1 -20749.118,E2 -20749.118} C_VEL
LIN {X 0,Y 213.748,Z 288.671,A -85,B 0,C 180,E1 -20753.713,E2 -20753.713} C_VEL
LIN {X 0,Y 213.79,Z 288.665,A -85,B 0,C 180,E1 -20758.724,E2 -20758.724} C_VEL
LIN {X 0,Y 213.82,Z 288.658,A -85,B 0,C 180,E1 -20762.602,E2 -20762.602} C_VEL
LIN {X 0,Y 213.846,Z 288.658,A -85,B 0,C 180,E1 -20766.952,E2 -20766.952} C_VEL
LIN {X 0,Y 213.937,Z 288.644,A -85,B 0,C 180,E1 -20772.803,E2 -20772.803} C_VEL
LIN {X 0,Y 213.974,Z 288.642,A -85,B 0,C 180,E1 -20776.708,E2 -20776.708} C_VEL
LIN {X 0,Y 214.161,Z 288.616,A -85,B 0,C 180,E1 -20780.556,E2 -20780.556} C_VEL
LIN {X 0,Y 214.221,Z 288.611,A -85,B 0,C 180,E1 -20782.459,E2 -20782.459} C_VEL
LIN {X 0,Y 214.438,Z 288.582,A -85,B 0,C 180,E1 -20788.121,E2 -20788.121} C_VEL
LIN {X 0,Y 214.543,Z 288.573,A -85,B 0,C 180,E1 -20790,E2 -20790} C_VEL
LIN {X 0,Y 214.438,Z 288.588,A -85,B 0,C 180,E1 -20791.878,E2 -20791.878} C_VEL
LIN {X 0,Y 214.219,Z 288.61,A -85,B 0,C 180,E1 -20797.54,E2 -20797.54} C_VEL
LIN {X 0,Y 214.037,Z 288.635,A -85,B 0,C 180,E1 -20801.362,E2 -20801.362} C_VEL
LIN {X 0,Y 213.926,Z 288.647,A -85,B 0,C 180,E1 -20805.237,E2 -20805.237} C_VEL
LIN {X 0,Y 213.828,Z 288.66,A -85,B 0,C 180,E1 -20809.187,E2 -20809.187} C_VEL
LIN {X 0,Y 213.866,Z 288.656,A -85,B 0,C 180,E1 -20814.575,E2 -20814.575} C_VEL
LIN {X 0,Y 221.008,Z 310.052,A -85,B 0,C 180,E1 -20816.016,E2 -20816.016} C_VEL
LIN {X 0,Y 219.3,Z 359.702,A -85,B 0,C 180,E1 -20817.978,E2 -20817.978} C_VEL
LIN {X 0,Y 218.709,Z 371.918,A -85,B 0,C 180,E1 -20818.816,E2 -20818.816} C_VEL
LIN {X 0,Y 217.835,Z 382.781,A -85,B 0,C 180,E1 -20819.948,E2 -20819.948} C_VEL
LIN {X 0,Y 217.002,Z 391.988,A -85,B 0,C 180,E1 -20821.21,E2 -20821.21} C_VEL
LIN {X 0,Y 216.072,Z 400.917,A -85,B 0,C 180,E1 -20822.752,E2 -20822.752} C_VEL
LIN {X 0,Y 214.759,Z 410.447,A -85,B 0,C 180,E1 -20824.834,E2 -20824.834} C_VEL
LIN {X 0,Y 213.798,Z 418.142,A -85,B 0,C 180,E1 -20827.011,E2 -20827.011} C_VEL
LIN {X 0,Y 213.091,Z 423.371,A -85,B 0,C 180,E1 -20828.801,E2 -20828.801} C_VEL
LIN {X 0,Y 212.596,Z 427.595,A -85,B 0,C 180,E1 -20830.509,E2 -20830.509} C_VEL
LIN {X 0,Y 212.242,Z 431.346,A -85,B 0,C 180,E1 -20832.316,E2 -20832.316} C_VEL
LIN {X 0,Y 211.71,Z 435.619,A -85,B 0,C 180,E1 -20834.977,E2 -20834.977} C_VEL
LIN {X 0,Y 211.51,Z 438.094,A -85,B 0,C 180,E1 -20836.969,E2 -20836.969} C_VEL
LIN {X 0,Y 211.536,Z 440.466,A -85,B 0,C 180,E1 -20839.829,E2 -20839.829} C_VEL
LIN {X 0,Y 212.093,Z 441.855,A -85,B 0,C 180,E1 -20843.386,E2 -20843.386} C_VEL
LIN {X 0,Y 212.822,Z 441.769,A -85,B 0,C 180,E1 -20845.85,E2 -20845.85} C_VEL
LIN {X 0,Y 213.988,Z 440.666,A -85,B 0,C 180,E1 -20848.638,E2 -20848.638} C_VEL
LIN {X 0,Y 215.648,Z 438.088,A -85,B 0,C 180,E1 -20851.631,E2 -20851.631} C_VEL
LIN {X 0,Y 217.239,Z 435.179,A -85,B 0,C 180,E1 -20853.884,E2 -20853.884} C_VEL
LIN {X 0,Y 219.319,Z 430.759,A -85,B 0,C 180,E1 -20856.389,E2 -20856.389} C_VEL
LIN {X 0,Y 221.072,Z 426.956,A -85,B 0,C 180,E1 -20858.088,E2 -20858.088} C_VEL
LIN {X 0,Y 223.479,Z 421.141,A -85,B 0,C 180,E1 -20860.165,E2 -20860.165} C_VEL
LIN {X 0,Y 225.567,Z 415.35,A -85,B 0,C 180,E1 -20861.848,E2 -20861.848} C_VEL
LIN {X 0,Y 227.848,Z 408.565,A -85,B 0,C 180,E1 -20863.441,E2 -20863.441} C_VEL
LIN {X 0,Y 230.07,Z 400.708,A -85,B 0,C 180,E1 -20864.952,E2 -20864.952} C_VEL
LIN {X 0,Y 232.549,Z 390.706,A -85,B 0,C 180,E1 -20866.456,E2 -20866.456} C_VEL
LIN {X 0,Y 234.597,Z 379.63,A -85,B 0,C 180,E1 -20867.677,E2 -20867.677} C_VEL
LIN {X 0,Y 235.878,Z 369.978,A -85,B 0,C 180,E1 -20868.472,E2 -20868.472} C_VEL
LIN {X 0,Y 236.857,Z 359.614,A -85,B 0,C 180,E1 -20869.059,E2 -20869.059} C_VEL
LIN {X 0,Y 238.88,Z 328.506,A -85,B 0,C 180,E1 -20870.247,E2 -20870.247} C_VEL
LIN {X 0,Y 234.683,Z 320.233,A -85,B 0,C 180,E1 -20871.689,E2 -20871.689} C_VEL
LIN {X 0,Y 228.656,Z 309.859,A -85,B 0,C 180,E1 -20873.881,E2 -20873.881} C_VEL
LIN {X 0,Y 224.232,Z 303.186,A -85,B 0,C 180,E1 -20875.608,E2 -20875.608} C_VEL
LIN {X 0,Y 221.735,Z 299.765,A -85,B 0,C 180,E1 -20876.651,E2 -20876.651} C_VEL
LIN {X 0,Y 220.735,Z 298.351,A -85,B 0,C 180,E1 -20877.093,E2 -20877.093} C_VEL
LIN {X 0,Y 218.521,Z 295.229,A -85,B 0,C 180,E1 -20878.101,E2 -20878.101} C_VEL
LIN {X 0,Y 217.81,Z 293.736,A -85,B 0,C 180,E1 -20878.475,E2 -20878.475} C_VEL
LIN {X 0,Y 215.722,Z 291.761,A -85,B 0,C 180,E1 -20879.424,E2 -20879.424} C_VEL
LIN {X 0,Y 214.658,Z 289.261,A -85,B 0,C 180,E1 -20880.06,E2 -20880.06} C_VEL
LIN {X 0,Y 214.531,Z 288.569,A -85,B 0,C 180,E1 -20880.236,E2 -20880.236} C_VEL
LIN {X 0,Y 214.135,Z 288.616,A -85,B 0,C 180,E1 -20883.765,E2 -20883.765} C_VEL
LIN {X 0,Y 214.223,Z 288.604,A -85,B 0,C 180,E1 -20887.542,E2 -20887.542} C_VEL
LIN {X 0,Y 214.018,Z 288.631,A -85,B 0,C 180,E1 -20891.365,E2 -20891.365} C_VEL
LIN {X 0,Y 213.926,Z 288.645,A -85,B 0,C 180,E1 -20895.239,E2 -20895.239} C_VEL
LIN {X 0,Y 213.864,Z 288.656,A -85,B 0,C 180,E1 -20899.186,E2 -20899.186} C_VEL
LIN {X 0,Y 213.845,Z 288.659,A -85,B 0,C 180,E1 -20903.229,E2 -20903.229} C_VEL
LIN {X 0,Y 213.827,Z 288.662,A -85,B 0,C 180,E1 -20907.452,E2 -20907.452} C_VEL
LIN {X 0,Y 213.778,Z 288.669,A -85,B 0,C 180,E1 -20911.737,E2 -20911.737} C_VEL
LIN {X 0,Y 213.753,Z 288.666,A -85,B 0,C 180,E1 -20916.288,E2 -20916.288} C_VEL
LIN {X 0,Y 213.748,Z 288.665,A -85,B 0,C 180,E1 -20921.118,E2 -20921.118} C_VEL
LIN {X 0,Y 213.838,Z 288.876,A -85,B 0,C 180,E1 -20922.041,E2 -20922.041} C_VEL
LIN {X 0,Y 215.634,Z 294.728,A -85,B 0,C 180,E1 -20926.81,E2 -20926.81} C_VEL
LIN {X 0,Y 215.96,Z 295.822,A -85,B 0,C 180,E1 -20927.61,E2 -20927.61} C_VEL
LIN {X 0,Y 216.271,Z 297.865,A -85,B 0,C 180,E1 -20928.491,E2 -20928.491} C_VEL
LIN {X 0,Y 216.453,Z 300.828,A -85,B 0,C 180,E1 -20929.196,E2 -20929.196} C_VEL
LIN {X 0,Y 217.283,Z 309.011,A -85,B 0,C 180,E1 -20930.514,E2 -20930.514} C_VEL
LIN {X 0,Y 218.304,Z 312.245,A -85,B 0,C 180,E1 -20931.136,E2 -20931.136} C_VEL
LIN {X 0,Y 221.022,Z 317.175,A -85,B 0,C 180,E1 -20932.389,E2 -20932.389} C_VEL
LIN {X 0,Y 225.583,Z 326.114,A -85,B 0,C 180,E1 -20934.334,E2 -20934.334} C_VEL
LIN {X 0,Y 229.268,Z 334.749,A -85,B 0,C 180,E1 -20935.861,E2 -20935.861} C_VEL
LIN {X 0,Y 231.12,Z 348.817,A -85,B 0,C 180,E1 -20937.109,E2 -20937.109} C_VEL
LIN {X 0,Y 232.022,Z 360.706,A -85,B 0,C 180,E1 -20937.971,E2 -20937.971} C_VEL
LIN {X 0,Y 230.337,Z 381.992,A -85,B 0,C 180,E1 -20938.816,E2 -20938.816} C_VEL
LIN {X 0,Y 228.535,Z 393.968,A -85,B 0,C 180,E1 -20939.571,E2 -20939.571} C_VEL
LIN {X 0,Y 226.581,Z 403.574,A -85,B 0,C 180,E1 -20940.457,E2 -20940.457} C_VEL
LIN {X 0,Y 224.125,Z 413.318,A -85,B 0,C 180,E1 -20941.637,E2 -20941.637} C_VEL
LIN {X 0,Y 222.07,Z 420.242,A -85,B 0,C 180,E1 -20942.685,E2 -20942.685} C_VEL
LIN {X 0,Y 219.578,Z 427.994,A -85,B 0,C 180,E1 -20944.146,E2 -20944.146} C_VEL
LIN {X 0,Y 216.627,Z 436.188,A -85,B 0,C 180,E1 -20946.076,E2 -20946.076} C_VEL
LIN {X 0,Y 213.669,Z 443.503,A -85,B 0,C 180,E1 -20948.283,E2 -20948.283} C_VEL
LIN {X 0,Y 211.114,Z 449.298,A -85,B 0,C 180,E1 -20950.556,E2 -20950.556} C_VEL
LIN {X 0,Y 209.341,Z 453.159,A -85,B 0,C 180,E1 -20952.414,E2 -20952.414} C_VEL
LIN {X 0,Y 207.311,Z 457.62,A -85,B 0,C 180,E1 -20955.271,E2 -20955.271} C_VEL
LIN {X 0,Y 205.839,Z 460.842,A -85,B 0,C 180,E1 -20958.179,E2 -20958.179} C_VEL
LIN {X 0,Y 205.167,Z 462.348,A -85,B 0,C 180,E1 -20960.139,E2 -20960.139} C_VEL
LIN {X 0,Y 204.751,Z 463.387,A -85,B 0,C 180,E1 -20962.109,E2 -20962.109} C_VEL
LIN {X 0,Y 204.547,Z 463.886,A -85,B 0,C 180,E1 -20965.153,E2 -20965.153} C_VEL
LIN {X 0,Y 204.674,Z 463.285,A -85,B 0,C 180,E1 -20968.033,E2 -20968.033} C_VEL
LIN {X 0,Y 204.775,Z 462.281,A -85,B 0,C 180,E1 -20970,E2 -20970} C_VEL
LIN {X 0,Y 204.752,Z 460.699,A -85,B 0,C 180,E1 -20971.967,E2 -20971.967} C_VEL
LIN {X 0,Y 204.748,Z 457.548,A -85,B 0,C 180,E1 -20974.635,E2 -20974.635} C_VEL
LIN {X 0,Y 204.845,Z 453.951,A -85,B 0,C 180,E1 -20976.897,E2 -20976.897} C_VEL
LIN {X 0,Y 205.148,Z 448.873,A -85,B 0,C 180,E1 -20979.365,E2 -20979.365} C_VEL
LIN {X 0,Y 205.586,Z 443.892,A -85,B 0,C 180,E1 -20981.336,E2 -20981.336} C_VEL
LIN {X 0,Y 206.29,Z 437.877,A -85,B 0,C 180,E1 -20983.295,E2 -20983.295} C_VEL
LIN {X 0,Y 207.189,Z 430.543,A -85,B 0,C 180,E1 -20985.242,E2 -20985.242} C_VEL
LIN {X 0,Y 208.244,Z 422.743,A -85,B 0,C 180,E1 -20986.923,E2 -20986.923} C_VEL
LIN {X 0,Y 209.022,Z 416.023,A -85,B 0,C 180,E1 -20988.121,E2 -20988.121} C_VEL
LIN {X 0,Y 209.945,Z 407.905,A -85,B 0,C 180,E1 -20989.303,E2 -20989.303} C_VEL
LIN {X 0,Y 210.994,Z 398.719,A -85,B 0,C 180,E1 -20990.344,E2 -20990.344} C_VEL
LIN {X 0,Y 211.822,Z 388.342,A -85,B 0,C 180,E1 -20991.214,E2 -20991.214} C_VEL
LIN {X 0,Y 212.457,Z 373.914,A -85,B 0,C 180,E1 -20991.95,E2 -20991.95} C_VEL
LIN {X 0,Y 213.017,Z 354.192,A -85,B 0,C 180,E1 -20992.744,E2 -20992.744} C_VEL
LIN {X 0,Y 208.799,Z 304.657,A -85,B 0,C 180,E1 -20995.168,E2 -20995.168} C_VEL
LIN {X 0,Y 209.164,Z 301.728,A -85,B 0,C 180,E1 -20996.436,E2 -20996.436} C_VEL
LIN {X 0,Y 207.462,Z 292.842,A -85,B 0,C 180,E1 -21000.54,E2 -21000.54} C_VEL
LIN {X 0,Y 206.83,Z 289.536,A -85,B 0,C 180,E1 -21002.15,E2 -21002.15} C_VEL
LIN {X 0,Y 206.702,Z 289.551,A -85,B 0,C 180,E1 -21007.735,E2 -21007.735} C_VEL
LIN {X 0,Y 206.649,Z 289.555,A -85,B 0,C 180,E1 -21011.563,E2 -21011.563} C_VEL
LIN {X 0,Y 206.634,Z 289.559,A -85,B 0,C 180,E1 -21015.581,E2 -21015.581} C_VEL
LIN {X 0,Y 206.662,Z 289.553,A -85,B 0,C 180,E1 -21019.747,E2 -21019.747} C_VEL
LIN {X 0,Y 206.701,Z 289.548,A -85,B 0,C 180,E1 -21024.687,E2 -21024.687} C_VEL
LIN {X 0,Y 206.716,Z 289.546,A -85,B 0,C 180,E1 -21029.336,E2 -21029.336} C_VEL
LIN {X 0,Y 206.734,Z 289.547,A -85,B 0,C 180,E1 -21033.771,E2 -21033.771} C_VEL
LIN {X 0,Y 206.758,Z 289.538,A -85,B 0,C 180,E1 -21038.042,E2 -21038.042} C_VEL
LIN {X 0,Y 206.873,Z 289.527,A -85,B 0,C 180,E1 -21042.195,E2 -21042.195} C_VEL
LIN {X 0,Y 206.893,Z 289.521,A -85,B 0,C 180,E1 -21046.243,E2 -21046.243} C_VEL
LIN {X 0,Y 207.099,Z 289.499,A -85,B 0,C 180,E1 -21050.229,E2 -21050.229} C_VEL
LIN {X 0,Y 207.06,Z 289.501,A -85,B 0,C 180,E1 -21054.154,E2 -21054.154} C_VEL
LIN {X 0,Y 207.38,Z 289.465,A -85,B 0,C 180,E1 -21058.056,E2 -21058.056} C_VEL
LIN {X 0,Y 207.513,Z 289.448,A -85,B 0,C 180,E1 -21059.998,E2 -21059.998} C_VEL
LIN {X 0,Y 207.38,Z 289.463,A -85,B 0,C 180,E1 -21061.94,E2 -21061.94} C_VEL
LIN {X 0,Y 207.175,Z 289.492,A -85,B 0,C 180,E1 -21067.797,E2 -21067.797} C_VEL
LIN {X 0,Y 206.94,Z 289.517,A -85,B 0,C 180,E1 -21071.756,E2 -21071.756} C_VEL
LIN {X 0,Y 206.863,Z 289.531,A -85,B 0,C 180,E1 -21075.769,E2 -21075.769} C_VEL
LIN {X 0,Y 206.809,Z 289.533,A -85,B 0,C 180,E1 -21079.865,E2 -21079.865} C_VEL
LIN {X 0,Y 206.764,Z 289.542,A -85,B 0,C 180,E1 -21084.07,E2 -21084.07} C_VEL
LIN {X 0,Y 206.74,Z 289.54,A -85,B 0,C 180,E1 -21088.417,E2 -21088.417} C_VEL
LIN {X 0,Y 206.705,Z 289.548,A -85,B 0,C 180,E1 -21092.954,E2 -21092.954} C_VEL
LIN {X 0,Y 206.717,Z 289.545,A -85,B 0,C 180,E1 -21097.729,E2 -21097.729} C_VEL
LIN {X 0,Y 206.701,Z 289.548,A -85,B 0,C 180,E1 -21102.842,E2 -21102.842} C_VEL
LIN {X 0,Y 206.71,Z 289.544,A -85,B 0,C 180,E1 -21107.158,E2 -21107.158} C_VEL
LIN {X 0,Y 206.754,Z 289.543,A -85,B 0,C 180,E1 -21111.424,E2 -21111.424} C_VEL
LIN {X 0,Y 206.725,Z 289.541,A -85,B 0,C 180,E1 -21114.694,E2 -21114.694} C_VEL
LIN {X 0,Y 206.718,Z 289.547,A -85,B 0,C 180,E1 -21119.338,E2 -21119.338} C_VEL
LIN {X 0,Y 206.727,Z 289.544,A -85,B 0,C 180,E1 -21123.771,E2 -21123.771} C_VEL
LIN {X 0,Y 206.751,Z 289.544,A -85,B 0,C 180,E1 -21128.043,E2 -21128.043} C_VEL
LIN {X 0,Y 206.867,Z 289.526,A -85,B 0,C 180,E1 -21132.196,E2 -21132.196} C_VEL
LIN {X 0,Y 206.907,Z 289.523,A -85,B 0,C 180,E1 -21136.245,E2 -21136.245} C_VEL
LIN {X 0,Y 207.099,Z 289.497,A -85,B 0,C 180,E1 -21140.231,E2 -21140.231} C_VEL
LIN {X 0,Y 207.161,Z 289.492,A -85,B 0,C 180,E1 -21142.201,E2 -21142.201} C_VEL
LIN {X 0,Y 207.374,Z 289.462,A -85,B 0,C 180,E1 -21148.057,E2 -21148.057} C_VEL
LIN {X 0,Y 207.508,Z 289.449,A -85,B 0,C 180,E1 -21150,E2 -21150} C_VEL
LIN {X 0,Y 207.374,Z 289.467,A -85,B 0,C 180,E1 -21151.942,E2 -21151.942} C_VEL
LIN {X 0,Y 207.159,Z 289.49,A -85,B 0,C 180,E1 -21157.799,E2 -21157.799} C_VEL
LIN {X 0,Y 206.974,Z 289.517,A -85,B 0,C 180,E1 -21161.755,E2 -21161.755} C_VEL
LIN {X 0,Y 206.86,Z 289.53,A -85,B 0,C 180,E1 -21165.77,E2 -21165.77} C_VEL
LIN {X 0,Y 206.772,Z 289.543,A -85,B 0,C 180,E1 -21169.869,E2 -21169.869} C_VEL
LIN {X 0,Y 206.797,Z 289.539,A -85,B 0,C 180,E1 -21174.067,E2 -21174.067} C_VEL
LIN {X 0,Y 214.236,Z 311.836,A -85,B 0,C 180,E1 -21175.618,E2 -21175.618} C_VEL
LIN {X 0,Y 212.41,Z 359.501,A -85,B 0,C 180,E1 -21177.552,E2 -21177.552} C_VEL
LIN {X 0,Y 211.851,Z 371.152,A -85,B 0,C 180,E1 -21178.346,E2 -21178.346} C_VEL
LIN {X 0,Y 210.888,Z 382.836,A -85,B 0,C 180,E1 -21179.572,E2 -21179.572} C_VEL
LIN {X 0,Y 210.145,Z 390.78,A -85,B 0,C 180,E1 -21180.663,E2 -21180.663} C_VEL
LIN {X 0,Y 209.245,Z 399.796,A -85,B 0,C 180,E1 -21182.221,E2 -21182.221} C_VEL
LIN {X 0,Y 208.157,Z 407.601,A -85,B 0,C 180,E1 -21183.879,E2 -21183.879} C_VEL
LIN {X 0,Y 207.071,Z 415.703,A -85,B 0,C 180,E1 -21186.005,E2 -21186.005} C_VEL
LIN {X 0,Y 206.152,Z 422.775,A -85,B 0,C 180,E1 -21188.366,E2 -21188.366} C_VEL
LIN {X 0,Y 205.488,Z 427.977,A -85,B 0,C 180,E1 -21190.527,E2 -21190.527} C_VEL
LIN {X 0,Y 205.145,Z 431.599,A -85,B 0,C 180,E1 -21192.326,E2 -21192.326} C_VEL
LIN {X 0,Y 204.596,Z 435.963,A -85,B 0,C 180,E1 -21195.12,E2 -21195.12} C_VEL
LIN {X 0,Y 204.37,Z 439.085,A -85,B 0,C 180,E1 -21197.892,E2 -21197.892} C_VEL
LIN {X 0,Y 204.422,Z 440.261,A -85,B 0,C 180,E1 -21199.218,E2 -21199.218} C_VEL
LIN {X 0,Y 204.729,Z 441.886,A -85,B 0,C 180,E1 -21202.141,E2 -21202.141} C_VEL
LIN {X 0,Y 205.479,Z 442.331,A -85,B 0,C 180,E1 -21205.17,E2 -21205.17} C_VEL
LIN {X 0,Y 206.124,Z 442.116,A -85,B 0,C 180,E1 -21206.941,E2 -21206.941} C_VEL
LIN {X 0,Y 207.278,Z 441.014,A -85,B 0,C 180,E1 -21209.432,E2 -21209.432} C_VEL
LIN {X 0,Y 208.651,Z 439.099,A -85,B 0,C 180,E1 -21211.866,E2 -21211.866} C_VEL
LIN {X 0,Y 210.457,Z 436.15,A -85,B 0,C 180,E1 -21214.371,E2 -21214.371} C_VEL
LIN {X 0,Y 212.327,Z 432.597,A -85,B 0,C 180,E1 -21216.599,E2 -21216.599} C_VEL
LIN {X 0,Y 215.161,Z 426.715,A -85,B 0,C 180,E1 -21219.309,E2 -21219.309} C_VEL
LIN {X 0,Y 217.403,Z 421.635,A -85,B 0,C 180,E1 -21221.141,E2 -21221.141} C_VEL
LIN {X 0,Y 219.504,Z 416.166,A -85,B 0,C 180,E1 -21222.776,E2 -21222.776} C_VEL
LIN {X 0,Y 221.88,Z 409.525,A -85,B 0,C 180,E1 -21224.383,E2 -21224.383} C_VEL
LIN {X 0,Y 224.132,Z 402.113,A -85,B 0,C 180,E1 -21225.863,E2 -21225.863} C_VEL
LIN {X 0,Y 226.469,Z 393.35,A -85,B 0,C 180,E1 -21227.26,E2 -21227.26} C_VEL
LIN {X 0,Y 228.821,Z 382.579,A -85,B 0,C 180,E1 -21228.577,E2 -21228.577} C_VEL
LIN {X 0,Y 230.418,Z 371.843,A -85,B 0,C 180,E1 -21229.527,E2 -21229.527} C_VEL
LIN {X 0,Y 231.451,Z 362.359,A -85,B 0,C 180,E1 -21230.112,E2 -21230.112} C_VEL
LIN {X 0,Y 233.628,Z 331.1,A -85,B 0,C 180,E1 -21231.351,E2 -21231.351} C_VEL
LIN {X 0,Y 228.16,Z 320.741,A -85,B 0,C 180,E1 -21233.368,E2 -21233.368} C_VEL
LIN {X 0,Y 223.106,Z 312.149,A -85,B 0,C 180,E1 -21235.388,E2 -21235.388} C_VEL
LIN {X 0,Y 220.423,Z 308.316,A -85,B 0,C 180,E1 -21236.517,E2 -21236.517} C_VEL
LIN {X 0,Y 217.369,Z 303.88,A -85,B 0,C 180,E1 -21237.903,E2 -21237.903} C_VEL
LIN {X 0,Y 215.002,Z 300.2,A -85,B 0,C 180,E1 -21239.065,E2 -21239.065} C_VEL
LIN {X 0,Y 212.269,Z 296.698,A -85,B 0,C 180,E1 -21240.476,E2 -21240.476} C_VEL
LIN {X 0,Y 211.497,Z 294.994,A -85,B 0,C 180,E1 -21240.955,E2 -21240.955} C_VEL
LIN {X 0,Y 208.703,Z 292.929,A -85,B 0,C 180,E1 -21242.414,E2 -21242.414} C_VEL
LIN {X 0,Y 207.327,Z 290.462,A -85,B 0,C 180,E1 -21243.342,E2 -21243.342} C_VEL
LIN {X 0,Y 207.127,Z 289.49,A -85,B 0,C 180,E1 -21243.588,E2 -21243.588} C_VEL
LIN {X 0,Y 207.163,Z 289.482,A -85,B 0,C 180,E1 -21247.801,E2 -21247.801} C_VEL
LIN {X 0,Y 206.938,Z 289.509,A -85,B 0,C 180,E1 -21251.759,E2 -21251.759} C_VEL
LIN {X 0,Y 206.86,Z 289.52,A -85,B 0,C 180,E1 -21255.773,E2 -21255.773} C_VEL
LIN {X 0,Y 206.796,Z 289.528,A -85,B 0,C 180,E1 -21259.869,E2 -21259.869} C_VEL
LIN {X 0,Y 206.761,Z 289.533,A -85,B 0,C 180,E1 -21264.074,E2 -21264.074} C_VEL
LIN {X 0,Y 206.743,Z 289.536,A -85,B 0,C 180,E1 -21268.421,E2 -21268.421} C_VEL
LIN {X 0,Y 206.708,Z 289.539,A -85,B 0,C 180,E1 -21272.958,E2 -21272.958} C_VEL
LIN {X 0,Y 206.721,Z 289.549,A -85,B 0,C 180,E1 -21275.322,E2 -21275.322} C_VEL
LIN {X 0,Y 206.691,Z 289.558,A -85,B 0,C 180,E1 -21278.852,E2 -21278.852} C_VEL
LIN {X 0,Y 207.89,Z 293.224,A -85,B 0,C 180,E1 -21282.543,E2 -21282.543} C_VEL
LIN {X 0,Y 209.395,Z 297.929,A -85,B 0,C 180,E1 -21286.449,E2 -21286.449} C_VEL
LIN {X 0,Y 212.314,Z 302.747,A -85,B 0,C 180,E1 -21288.144,E2 -21288.144} C_VEL
LIN {X 0,Y 214.055,Z 305.126,A -85,B 0,C 180,E1 -21289.04,E2 -21289.04} C_VEL
LIN {X 0,Y 218.034,Z 311.737,A -85,B 0,C 180,E1 -21291.005,E2 -21291.005} C_VEL
LIN {X 0,Y 218.304,Z 312.245,A -85,B 0,C 180,E1 -21291.136,E2 -21291.136} C_VEL
LIN {X 0,Y 221.115,Z 319.956,A -85,B 0,C 180,E1 -21292.596,E2 -21292.596} C_VEL
LIN {X 0,Y 222.417,Z 325.052,A -85,B 0,C 180,E1 -21293.328,E2 -21293.328} C_VEL
LIN {X 0,Y 223.794,Z 332.215,A -85,B 0,C 180,E1 -21294.184,E2 -21294.184} C_VEL
LIN {X 0,Y 224.85,Z 339.595,A -85,B 0,C 180,E1 -21294.942,E2 -21294.942} C_VEL
LIN {X 0,Y 226.34,Z 353.676,A -85,B 0,C 180,E1 -21296.184,E2 -21296.184} C_VEL
LIN {X 0,Y 226.832,Z 362.337,A -85,B 0,C 180,E1 -21296.8,E2 -21296.8} C_VEL
LIN {X 0,Y 225.139,Z 382.227,A -85,B 0,C 180,E1 -21297.604,E2 -21297.604} C_VEL
LIN {X 0,Y 223.096,Z 394.66,A -85,B 0,C 180,E1 -21298.429,E2 -21298.429} C_VEL
LIN {X 0,Y 220.904,Z 404.714,A -85,B 0,C 180,E1 -21299.402,E2 -21299.402} C_VEL
LIN {X 0,Y 218.749,Z 412.715,A -85,B 0,C 180,E1 -21300.399,E2 -21300.399} C_VEL
LIN {X 0,Y 216.254,Z 420.598,A -85,B 0,C 180,E1 -21301.623,E2 -21301.623} C_VEL
LIN {X 0,Y 213.282,Z 429.193,A -85,B 0,C 180,E1 -21303.324,E2 -21303.324} C_VEL
LIN {X 0,Y 209.555,Z 438.497,A -85,B 0,C 180,E1 -21305.744,E2 -21305.744} C_VEL
LIN {X 0,Y 207.131,Z 444.006,A -85,B 0,C 180,E1 -21307.561,E2 -21307.561} C_VEL
LIN {X 0,Y 204.449,Z 449.634,A -85,B 0,C 180,E1 -21309.895,E2 -21309.895} C_VEL
LIN {X 0,Y 201.839,Z 454.931,A -85,B 0,C 180,E1 -21312.785,E2 -21312.785} C_VEL
LIN {X 0,Y 199.867,Z 458.881,A -85,B 0,C 180,E1 -21315.751,E2 -21315.751} C_VEL
LIN {X 0,Y 198.88,Z 460.736,A -85,B 0,C 180,E1 -21317.76,E2 -21317.76} C_VEL
LIN {X 0,Y 198.168,Z 462.116,A -85,B 0,C 180,E1 -21319.787,E2 -21319.787} C_VEL
LIN {X 0,Y 197.703,Z 463.041,A -85,B 0,C 180,E1 -21321.826,E2 -21321.826} C_VEL
LIN {X 0,Y 197.5,Z 463.488,A -85,B 0,C 180,E1 -21323.872,E2 -21323.872} C_VEL
LIN {X 0,Y 197.48,Z 463.339,A -85,B 0,C 180,E1 -21325.919,E2 -21325.919} C_VEL
LIN {X 0,Y 197.606,Z 462.707,A -85,B 0,C 180,E1 -21327.962,E2 -21327.962} C_VEL
LIN {X 0,Y 197.706,Z 461.584,A -85,B 0,C 180,E1 -21330,E2 -21330} C_VEL
LIN {X 0,Y 197.722,Z 458.79,A -85,B 0,C 180,E1 -21333.057,E2 -21333.057} C_VEL
LIN {X 0,Y 197.708,Z 455.522,A -85,B 0,C 180,E1 -21335.53,E2 -21335.53} C_VEL
LIN {X 0,Y 197.948,Z 449.965,A -85,B 0,C 180,E1 -21338.679,E2 -21338.679} C_VEL
LIN {X 0,Y 198.477,Z 443.963,A -85,B 0,C 180,E1 -21341.231,E2 -21341.231} C_VEL
LIN {X 0,Y 199.156,Z 438.048,A -85,B 0,C 180,E1 -21343.261,E2 -21343.261} C_VEL
LIN {X 0,Y 200.066,Z 430.841,A -85,B 0,C 180,E1 -21345.276,E2 -21345.276} C_VEL
LIN {X 0,Y 201.118,Z 423.192,A -85,B 0,C 180,E1 -21347.017,E2 -21347.017} C_VEL
LIN {X 0,Y 202.067,Z 415.158,A -85,B 0,C 180,E1 -21348.504,E2 -21348.504} C_VEL
LIN {X 0,Y 203.058,Z 406.948,A -85,B 0,C 180,E1 -21349.722,E2 -21349.722} C_VEL
LIN {X 0,Y 204.113,Z 397.602,A -85,B 0,C 180,E1 -21350.798,E2 -21350.798} C_VEL
LIN {X 0,Y 204.959,Z 386.098,A -85,B 0,C 180,E1 -21351.762,E2 -21351.762} C_VEL
LIN {X 0,Y 205.601,Z 371.216,A -85,B 0,C 180,E1 -21352.48,E2 -21352.48} C_VEL
LIN {X 0,Y 206.037,Z 353.979,A -85,B 0,C 180,E1 -21353.204,E2 -21353.204} C_VEL
LIN {X 0,Y 201.915,Z 304.169,A -85,B 0,C 180,E1 -21355.765,E2 -21355.765} C_VEL
LIN {X 0,Y 201.981,Z 301.7,A -85,B 0,C 180,E1 -21356.894,E2 -21356.894} C_VEL
LIN {X 0,Y 200.213,Z 292.771,A -85,B 0,C 180,E1 -21361.182,E2 -21361.182} C_VEL
LIN {X 0,Y 199.789,Z 290.413,A -85,B 0,C 180,E1 -21362.406,E2 -21362.406} C_VEL
LIN {X 0,Y 199.636,Z 290.427,A -85,B 0,C 180,E1 -21366.76,E2 -21366.76} C_VEL
LIN {X 0,Y 199.642,Z 290.43,A -85,B 0,C 180,E1 -21369.32,E2 -21369.32} C_VEL
LIN {X 0,Y 199.581,Z 290.433,A -85,B 0,C 180,E1 -21374.771,E2 -21374.771} C_VEL
LIN {X 0,Y 199.58,Z 290.436,A -85,B 0,C 180,E1 -21378.003,E2 -21378.003} C_VEL
LIN {X 0,Y 199.612,Z 290.429,A -85,B 0,C 180,E1 -21380.767,E2 -21380.767} C_VEL
LIN {X 0,Y 199.614,Z 290.434,A -85,B 0,C 180,E1 -21385.712,E2 -21385.712} C_VEL
LIN {X 0,Y 199.695,Z 290.42,A -85,B 0,C 180,E1 -21388.134,E2 -21388.134} C_VEL
LIN {X 0,Y 199.688,Z 290.421,A -85,B 0,C 180,E1 -21392.77,E2 -21392.77} C_VEL
LIN {X 0,Y 199.739,Z 290.415,A -85,B 0,C 180,E1 -21397.228,E2 -21397.228} C_VEL
LIN {X 0,Y 199.797,Z 290.411,A -85,B 0,C 180,E1 -21401.756,E2 -21401.756} C_VEL
LIN {X 0,Y 199.834,Z 290.402,A -85,B 0,C 180,E1 -21405.747,E2 -21405.747} C_VEL
LIN {X 0,Y 200.022,Z 290.382,A -85,B 0,C 180,E1 -21409.88,E2 -21409.88} C_VEL
LIN {X 0,Y 200.021,Z 290.379,A -85,B 0,C 180,E1 -21413.948,E2 -21413.948} C_VEL
LIN {X 0,Y 200.319,Z 290.345,A -85,B 0,C 180,E1 -21417.988,E2 -21417.988} C_VEL
LIN {X 0,Y 200.477,Z 290.325,A -85,B 0,C 180,E1 -21419.998,E2 -21419.998} C_VEL
LIN {X 0,Y 200.029,Z 290.378,A -85,B 0,C 180,E1 -21424.028,E2 -21424.028} C_VEL
LIN {X 0,Y 200.117,Z 290.37,A -85,B 0,C 180,E1 -21428.074,E2 -21428.074} C_VEL
LIN {X 0,Y 199.883,Z 290.394,A -85,B 0,C 180,E1 -21432.177,E2 -21432.177} C_VEL
LIN {X 0,Y 199.802,Z 290.408,A -85,B 0,C 180,E1 -21436.342,E2 -21436.342} C_VEL
LIN {X 0,Y 199.822,Z 290.404,A -85,B 0,C 180,E1 -21438.452,E2 -21438.452} C_VEL
LIN {X 0,Y 199.738,Z 290.418,A -85,B 0,C 180,E1 -21443.819,E2 -21443.819} C_VEL
LIN {X 0,Y 199.708,Z 290.416,A -85,B 0,C 180,E1 -21448.385,E2 -21448.385} C_VEL
LIN {X 0,Y 199.659,Z 290.426,A -85,B 0,C 180,E1 -21452.351,E2 -21452.351} C_VEL
LIN {X 0,Y 199.646,Z 290.424,A -85,B 0,C 180,E1 -21456.756,E2 -21456.756} C_VEL
LIN {X 0,Y 199.67,Z 290.423,A -85,B 0,C 180,E1 -21459.311,E2 -21459.311} C_VEL
LIN {X 0,Y 199.643,Z 290.428,A -85,B 0,C 180,E1 -21462.332,E2 -21462.332} C_VEL
LIN {X 0,Y 199.66,Z 290.424,A -85,B 0,C 180,E1 -21465.252,E2 -21465.252} C_VEL
LIN {X 0,Y 199.66,Z 290.426,A -85,B 0,C 180,E1 -21468.026,E2 -21468.026} C_VEL
LIN {X 0,Y 199.674,Z 290.423,A -85,B 0,C 180,E1 -21470.742,E2 -21470.742} C_VEL
LIN {X 0,Y 199.629,Z 290.428,A -85,B 0,C 180,E1 -21475.717,E2 -21475.717} C_VEL
LIN {X 0,Y 199.698,Z 290.422,A -85,B 0,C 180,E1 -21478.137,E2 -21478.137} C_VEL
LIN {X 0,Y 199.681,Z 290.419,A -85,B 0,C 180,E1 -21482.771,E2 -21482.771} C_VEL
LIN {X 0,Y 199.732,Z 290.417,A -85,B 0,C 180,E1 -21487.228,E2 -21487.228} C_VEL
LIN {X 0,Y 199.79,Z 290.408,A -85,B 0,C 180,E1 -21491.757,E2 -21491.757} C_VEL
LIN {X 0,Y 199.841,Z 290.406,A -85,B 0,C 180,E1 -21495.748,E2 -21495.748} C_VEL
LIN {X 0,Y 200.064,Z 290.374,A -85,B 0,C 180,E1 -21499.884,E2 -21499.884} C_VEL
LIN {X 0,Y 200.027,Z 290.382,A -85,B 0,C 180,E1 -21503.949,E2 -21503.949} C_VEL
LIN {X 0,Y 200.314,Z 290.342,A -85,B 0,C 180,E1 -21507.989,E2 -21507.989} C_VEL
LIN {X 0,Y 200.472,Z 290.325,A -85,B 0,C 180,E1 -21510,E2 -21510} C_VEL
LIN {X 0,Y 200.022,Z 290.382,A -85,B 0,C 180,E1 -21514.029,E2 -21514.029} C_VEL
LIN {X 0,Y 200.103,Z 290.371,A -85,B 0,C 180,E1 -21518.075,E2 -21518.075} C_VEL
LIN {X 0,Y 199.906,Z 290.396,A -85,B 0,C 180,E1 -21522.177,E2 -21522.177} C_VEL
LIN {X 0,Y 199.797,Z 290.409,A -85,B 0,C 180,E1 -21526.343,E2 -21526.343} C_VEL
LIN {X 0,Y 199.683,Z 290.423,A -85,B 0,C 180,E1 -21530.606,E2 -21530.606} C_VEL
LIN {X 0,Y 199.733,Z 290.418,A -85,B 0,C 180,E1 -21533.545,E2 -21533.545} C_VEL
LIN {X 0,Y 207.322,Z 312.984,A -85,B 0,C 180,E1 -21535.16,E2 -21535.16} C_VEL
LIN {X 0,Y 205.451,Z 360.242,A -85,B 0,C 180,E1 -21537.158,E2 -21537.158} C_VEL
LIN {X 0,Y 204.845,Z 372.249,A -85,B 0,C 180,E1 -21538.025,E2 -21538.025} C_VEL
LIN {X 0,Y 203.893,Z 383.127,A -85,B 0,C 180,E1 -21539.22,E2 -21539.22} C_VEL
LIN {X 0,Y 203.048,Z 392.163,A -85,B 0,C 180,E1 -21540.527,E2 -21540.527} C_VEL
LIN {X 0,Y 202.181,Z 400.36,A -85,B 0,C 180,E1 -21542.011,E2 -21542.011} C_VEL
LIN {X 0,Y 201.039,Z 408.337,A -85,B 0,C 180,E1 -21543.779,E2 -21543.779} C_VEL
LIN {X 0,Y 199.92,Z 416.597,A -85,B 0,C 180,E1 -21546.05,E2 -21546.05} C_VEL
LIN {X 0,Y 198.991,Z 423.318,A -85,B 0,C 180,E1 -21548.404,E2 -21548.404} C_VEL
LIN {X 0,Y 198.365,Z 428.603,A -85,B 0,C 180,E1 -21550.697,E2 -21550.697} C_VEL
LIN {X 0,Y 197.999,Z 431.937,A -85,B 0,C 180,E1 -21552.406,E2 -21552.406} C_VEL
LIN {X 0,Y 197.473,Z 436.421,A -85,B 0,C 180,E1 -21555.379,E2 -21555.379} C_VEL
LIN {X 0,Y 197.274,Z 439.685,A -85,B 0,C 180,E1 -21558.427,E2 -21558.427} C_VEL
LIN {X 0,Y 197.546,Z 441.784,A -85,B 0,C 180,E1 -21561.505,E2 -21561.505} C_VEL
LIN {X 0,Y 198.218,Z 442.75,A -85,B 0,C 180,E1 -21564.633,E2 -21564.633} C_VEL
LIN {X 0,Y 199.463,Z 442.364,A -85,B 0,C 180,E1 -21568.097,E2 -21568.097} C_VEL
LIN {X 0,Y 200.971,Z 440.885,A -85,B 0,C 180,E1 -21570.954,E2 -21570.954} C_VEL
LIN {X 0,Y 203.077,Z 437.948,A -85,B 0,C 180,E1 -21574.128,E2 -21574.128} C_VEL
LIN {X 0,Y 205.737,Z 433.542,A -85,B 0,C 180,E1 -21577.264,E2 -21577.264} C_VEL
LIN {X 0,Y 208.417,Z 428.479,A -85,B 0,C 180,E1 -21579.782,E2 -21579.782} C_VEL
LIN {X 0,Y 211.271,Z 422.439,A -85,B 0,C 180,E1 -21582.081,E2 -21582.081} C_VEL
LIN {X 0,Y 213.965,Z 415.925,A -85,B 0,C 180,E1 -21584.057,E2 -21584.057} C_VEL
LIN {X 0,Y 216.763,Z 408.384,A -85,B 0,C 180,E1 -21585.872,E2 -21585.872} C_VEL
LIN {X 0,Y 219.924,Z 398.26,A -85,B 0,C 180,E1 -21587.78,E2 -21587.78} C_VEL
LIN {X 0,Y 222.472,Z 387.918,A -85,B 0,C 180,E1 -21589.213,E2 -21589.213} C_VEL
LIN {X 0,Y 224.335,Z 378.392,A -85,B 0,C 180,E1 -21590.219,E2 -21590.219} C_VEL
LIN {X 0,Y 225.69,Z 368.918,A -85,B 0,C 180,E1 -21590.974,E2 -21590.974} C_VEL
LIN {X 0,Y 226.873,Z 356.342,A -85,B 0,C 180,E1 -21591.626,E2 -21591.626} C_VEL
LIN {X 0,Y 228.48,Z 333.884,A -85,B 0,C 180,E1 -21592.499,E2 -21592.499} C_VEL
LIN {X 0,Y 223.142,Z 323.68,A -85,B 0,C 180,E1 -21594.645,E2 -21594.645} C_VEL
LIN {X 0,Y 218.762,Z 316.231,A -85,B 0,C 180,E1 -21596.545,E2 -21596.545} C_VEL
LIN {X 0,Y 213.995,Z 309.324,A -85,B 0,C 180,E1 -21598.767,E2 -21598.767} C_VEL
LIN {X 0,Y 211.394,Z 305.298,A -85,B 0,C 180,E1 -21600.151,E2 -21600.151} C_VEL
LIN {X 0,Y 209.068,Z 301.886,A -85,B 0,C 180,E1 -21601.466,E2 -21601.466} C_VEL
LIN {X 0,Y 207.767,Z 300.605,A -85,B 0,C 180,E1 -21602.183,E2 -21602.183} C_VEL
LIN {X 0,Y 205.419,Z 297.972,A -85,B 0,C 180,E1 -21603.618,E2 -21603.618} C_VEL
LIN {X 0,Y 204.398,Z 296.079,A -85,B 0,C 180,E1 -21604.363,E2 -21604.363} C_VEL
LIN {X 0,Y 201.752,Z 294.191,A -85,B 0,C 180,E1 -21606.126,E2 -21606.126} C_VEL
LIN {X 0,Y 200.444,Z 291.929,A -85,B 0,C 180,E1 -21607.24,E2 -21607.24} C_VEL
LIN {X 0,Y 200.12,Z 290.359,A -85,B 0,C 180,E1 -21607.696,E2 -21607.696} C_VEL
LIN {X 0,Y 200.032,Z 290.382,A -85,B 0,C 180,E1 -21610.349,E2 -21610.349} C_VEL
LIN {X 0,Y 199.8,Z 290.396,A -85,B 0,C 180,E1 -21616.345,E2 -21616.345} C_VEL
LIN {X 0,Y 199.821,Z 290.403,A -85,B 0,C 180,E1 -21618.456,E2 -21618.456} C_VEL
LIN {X 0,Y 199.734,Z 290.41,A -85,B 0,C 180,E1 -21623.819,E2 -21623.819} C_VEL
LIN {X 0,Y 199.711,Z 290.411,A -85,B 0,C 180,E1 -21628.389,E2 -21628.389} C_VEL
LIN {X 0,Y 199.663,Z 290.42,A -85,B 0,C 180,E1 -21632.354,E2 -21632.354} C_VEL
LIN {X 0,Y 199.702,Z 290.557,A -85,B 0,C 180,E1 -21635.145,E2 -21635.145} C_VEL
LIN {X 0,Y 200.856,Z 294.221,A -85,B 0,C 180,E1 -21639.668,E2 -21639.668} C_VEL
LIN {X 0,Y 201.863,Z 296.863,A -85,B 0,C 180,E1 -21642.342,E2 -21642.342} C_VEL
LIN {X 0,Y 205.391,Z 302.391,A -85,B 0,C 180,E1 -21644.893,E2 -21644.893} C_VEL
LIN {X 0,Y 206.888,Z 304.414,A -85,B 0,C 180,E1 -21645.836,E2 -21645.836} C_VEL
LIN {X 0,Y 210.332,Z 309.758,A -85,B 0,C 180,E1 -21647.865,E2 -21647.865} C_VEL
LIN {X 0,Y 214.774,Z 317.312,A -85,B 0,C 180,E1 -21650.221,E2 -21650.221} C_VEL
LIN {X 0,Y 217.914,Z 323.323,A -85,B 0,C 180,E1 -21651.767,E2 -21651.767} C_VEL
LIN {X 0,Y 222.748,Z 333.409,A -85,B 0,C 180,E1 -21653.949,E2 -21653.949} C_VEL
LIN {X 0,Y 224.673,Z 338.376,A -85,B 0,C 180,E1 -21654.817,E2 -21654.817} C_VEL
LIN {X 0,Y 224.85,Z 339.595,A -85,B 0,C 180,E1 -21654.942,E2 -21654.942} C_VEL
LIN {X 0,Y 225.061,Z 345.288,A -85,B 0,C 180,E1 -21655.345,E2 -21655.345} C_VEL
LIN {X 0,Y 224.511,Z 351.166,A -85,B 0,C 180,E1 -21655.545,E2 -21655.545} C_VEL
LIN {X 0,Y 222.374,Z 363.072,A -85,B 0,C 180,E1 -21655.666,E2 -21655.666} C_VEL
LIN {X 0,Y 221.197,Z 371.063,A -85,B 0,C 180,E1 -21655.822,E2 -21655.822} C_VEL
LIN {X 0,Y 219.609,Z 385.363,A -85,B 0,C 180,E1 -21656.508,E2 -21656.508} C_VEL
LIN {X 0,Y 217.994,Z 394.213,A -85,B 0,C 180,E1 -21657.133,E2 -21657.133} C_VEL
LIN {X 0,Y 215.804,Z 403.879,A -85,B 0,C 180,E1 -21658.071,E2 -21658.071} C_VEL
LIN {X 0,Y 213.533,Z 411.862,A -85,B 0,C 180,E1 -21659.053,E2 -21659.053} C_VEL
LIN {X 0,Y 210.924,Z 419.818,A -85,B 0,C 180,E1 -21660.289,E2 -21660.289} C_VEL
LIN {X 0,Y 207.788,Z 428.474,A -85,B 0,C 180,E1 -21662.013,E2 -21662.013} C_VEL
LIN {X 0,Y 203.84,Z 437.853,A -85,B 0,C 180,E1 -21664.472,E2 -21664.472} C_VEL
LIN {X 0,Y 201.305,Z 443.365,A -85,B 0,C 180,E1 -21666.33,E2 -21666.33} C_VEL
LIN {X 0,Y 198.89,Z 448.024,A -85,B 0,C 180,E1 -21668.222,E2 -21668.222} C_VEL
LIN {X 0,Y 195.88,Z 453.539,A -85,B 0,C 180,E1 -21671.162,E2 -21671.162} C_VEL
LIN {X 0,Y 193.576,Z 457.711,A -85,B 0,C 180,E1 -21674.2,E2 -21674.2} C_VEL
LIN {X 0,Y 191.92,Z 460.653,A -85,B 0,C 180,E1 -21677.308,E2 -21677.308} C_VEL
LIN {X 0,Y 191.156,Z 461.9,A -85,B 0,C 180,E1 -21679.408,E2 -21679.408} C_VEL
LIN {X 0,Y 190.678,Z 462.698,A -85,B 0,C 180,E1 -21681.523,E2 -21681.523} C_VEL
LIN {X 0,Y 190.421,Z 463.053,A -85,B 0,C 180,E1 -21683.644,E2 -21683.644} C_VEL
LIN {X 0,Y 190.408,Z 462.877,A -85,B 0,C 180,E1 -21685.767,E2 -21685.767} C_VEL
LIN {X 0,Y 190.537,Z 462.131,A -85,B 0,C 180,E1 -21687.887,E2 -21687.887} C_VEL
LIN {X 0,Y 190.638,Z 460.888,A -85,B 0,C 180,E1 -21690.001,E2 -21690.001} C_VEL
LIN {X 0,Y 190.662,Z 457.969,A -85,B 0,C 180,E1 -21693.17,E2 -21693.17} C_VEL
LIN {X 0,Y 190.665,Z 453.662,A -85,B 0,C 180,E1 -21696.349,E2 -21696.349} C_VEL
LIN {X 0,Y 191.025,Z 447.586,A -85,B 0,C 180,E1 -21699.53,E2 -21699.53} C_VEL
LIN {X 0,Y 191.507,Z 442.517,A -85,B 0,C 180,E1 -21701.645,E2 -21701.645} C_VEL
LIN {X 0,Y 192.251,Z 436.397,A -85,B 0,C 180,E1 -21703.746,E2 -21703.746} C_VEL
LIN {X 0,Y 193.228,Z 428.946,A -85,B 0,C 180,E1 -21705.83,E2 -21705.83} C_VEL
LIN {X 0,Y 194.341,Z 421,A -85,B 0,C 180,E1 -21707.63,E2 -21707.63} C_VEL
LIN {X 0,Y 195.514,Z 411.09,A -85,B 0,C 180,E1 -21709.421,E2 -21709.421} C_VEL
LIN {X 0,Y 196.958,Z 399.696,A -85,B 0,C 180,E1 -21710.906,E2 -21710.906} C_VEL
LIN {X 0,Y 197.754,Z 389.896,A -85,B 0,C 180,E1 -21711.842,E2 -21711.842} C_VEL
LIN {X 0,Y 198.404,Z 379.479,A -85,B 0,C 180,E1 -21712.52,E2 -21712.52} C_VEL
LIN {X 0,Y 199.121,Z 354.198,A -85,B 0,C 180,E1 -21713.646,E2 -21713.646} C_VEL
LIN {X 0,Y 194.988,Z 303.805,A -85,B 0,C 180,E1 -21716.344,E2 -21716.344} C_VEL
LIN {X 0,Y 193.904,Z 297.249,A -85,B 0,C 180,E1 -21719.553,E2 -21719.553} C_VEL
LIN {X 0,Y 192.737,Z 291.291,A -85,B 0,C 180,E1 -21722.615,E2 -21722.615} C_VEL
LIN {X 0,Y 192.575,Z 291.308,A -85,B 0,C 180,E1 -21728.346,E2 -21728.346} C_VEL
LIN {X 0,Y 192.495,Z 291.315,A -85,B 0,C 180,E1 -21733.095,E2 -21733.095} C_VEL
LIN {X 0,Y 192.492,Z 291.318,A -85,B 0,C 180,E1 -21736.904,E2 -21736.904} C_VEL
LIN {X 0,Y 192.553,Z 291.309,A -85,B 0,C 180,E1 -21741.647,E2 -21741.647} C_VEL
LIN {X 0,Y 192.599,Z 291.305,A -85,B 0,C 180,E1 -21746.812,E2 -21746.812} C_VEL
LIN {X 0,Y 192.666,Z 291.297,A -85,B 0,C 180,E1 -21751.69,E2 -21751.69} C_VEL
LIN {X 0,Y 192.707,Z 291.29,A -85,B 0,C 180,E1 -21756.347,E2 -21756.347} C_VEL
LIN {X 0,Y 192.733,Z 291.29,A -85,B 0,C 180,E1 -21761.456,E2 -21761.456} C_VEL
LIN {X 0,Y 192.763,Z 291.285,A -85,B 0,C 180,E1 -21765.212,E2 -21765.212} C_VEL
LIN {X 0,Y 192.945,Z 291.263,A -85,B 0,C 180,E1 -21769.565,E2 -21769.565} C_VEL
LIN {X 0,Y 192.984,Z 291.257,A -85,B 0,C 180,E1 -21773.726,E2 -21773.726} C_VEL
LIN {X 0,Y 193.261,Z 291.224,A -85,B 0,C 180,E1 -21777.914,E2 -21777.914} C_VEL
LIN {X 0,Y 193.441,Z 291.201,A -85,B 0,C 180,E1 -21779.998,E2 -21779.998} C_VEL
LIN {X 0,Y 192.975,Z 291.256,A -85,B 0,C 180,E1 -21784.175,E2 -21784.175} C_VEL
LIN {X 0,Y 193.066,Z 291.247,A -85,B 0,C 180,E1 -21788.371,E2 -21788.371} C_VEL
LIN {X 0,Y 192.807,Z 291.275,A -85,B 0,C 180,E1 -21792.631,E2 -21792.631} C_VEL
LIN {X 0,Y 192.768,Z 291.284,A -85,B 0,C 180,E1 -21796.956,E2 -21796.956} C_VEL
LIN {X 0,Y 192.652,Z 291.296,A -85,B 0,C 180,E1 -21801.393,E2 -21801.393} C_VEL
LIN {X 0,Y 192.665,Z 291.297,A -85,B 0,C 180,E1 -21804.226,E2 -21804.226} C_VEL
LIN {X 0,Y 192.646,Z 291.296,A -85,B 0,C 180,E1 -21808.89,E2 -21808.89} C_VEL
LIN {X 0,Y 192.596,Z 291.306,A -85,B 0,C 180,E1 -21813.184,E2 -21813.184} C_VEL
LIN {X 0,Y 192.593,Z 291.303,A -85,B 0,C 180,E1 -21818.339,E2 -21818.339} C_VEL
LIN {X 0,Y 192.595,Z 291.306,A -85,B 0,C 180,E1 -21823.891,E2 -21823.891} C_VEL
LIN {X 0,Y 192.578,Z 291.307,A -85,B 0,C 180,E1 -21828.937,E2 -21828.937} C_VEL
LIN {X 0,Y 192.613,Z 291.303,A -85,B 0,C 180,E1 -21833.388,E2 -21833.388} C_VEL
LIN {X 0,Y 192.602,Z 291.304,A -85,B 0,C 180,E1 -21837.058,E2 -21837.058} C_VEL
LIN {X 0,Y 192.659,Z 291.298,A -85,B 0,C 180,E1 -21841.691,E2 -21841.691} C_VEL
LIN {X 0,Y 192.7,Z 291.293,A -85,B 0,C 180,E1 -21846.348,E2 -21846.348} C_VEL
LIN {X 0,Y 192.726,Z 291.288,A -85,B 0,C 180,E1 -21851.457,E2 -21851.457} C_VEL
LIN {X 0,Y 192.765,Z 291.284,A -85,B 0,C 180,E1 -21855.214,E2 -21855.214} C_VEL
LIN {X 0,Y 192.975,Z 291.258,A -85,B 0,C 180,E1 -21859.508,E2 -21859.508} C_VEL
LIN {X 0,Y 193.055,Z 291.247,A -85,B 0,C 180,E1 -21861.627,E2 -21861.627} C_VEL
LIN {X 0,Y 193.256,Z 291.221,A -85,B 0,C 180,E1 -21867.915,E2 -21867.915} C_VEL
LIN {X 0,Y 193.436,Z 291.201,A -85,B 0,C 180,E1 -21869.999,E2 -21869.999} C_VEL
LIN {X 0,Y 192.968,Z 291.259,A -85,B 0,C 180,E1 -21874.177,E2 -21874.177} C_VEL
LIN {X 0,Y 193.054,Z 291.247,A -85,B 0,C 180,E1 -21878.372,E2 -21878.372} C_VEL
LIN {X 0,Y 192.846,Z 291.274,A -85,B 0,C 180,E1 -21882.63,E2 -21882.63} C_VEL
LIN {X 0,Y 192.75,Z 291.286,A -85,B 0,C 180,E1 -21886.958,E2 -21886.958} C_VEL
LIN {X 0,Y 192.684,Z 291.295,A -85,B 0,C 180,E1 -21892.8,E2 -21892.8} C_VEL
